LIN {X 0,Y 742.952,Z 751.201,A -85,B 0,C 180,E1 34860.975,E2 34860.975} C_VEL
LIN {X 0,Y 742.857,Z 676.201,A -85,B 0,C 180,E1 34860.963,E2 34860.963} C_VEL
LIN {X 0,Y 740.648,Z 678.554,A -85,B 0,C 180,E1 34860.677,E2 34860.677} C_VEL
LIN {X 0,Y 736.693,Z 689.627,A -85,B 0,C 180,E1 34860.154,E2 34860.154} C_VEL
LIN {X 0,Y 733.637,Z 695.78,A -85,B 0,C 180,E1 34859.741,E2 34859.741} C_VEL
LIN {X 0,Y 731.906,Z 697.683,A -85,B 0,C 180,E1 34859.503,E2 34859.503} C_VEL
LIN {X 0,Y 730.902,Z 697.691,A -85,B 0,C 180,E1 34859.356,E2 34859.356} C_VEL
LIN {X 0,Y 730.384,Z 754.623,A -85,B 0,C 180,E1 34856.592,E2 34856.592} C_VEL
LIN {X 0,Y 730.458,Z 758.053,A -85,B 0,C 180,E1 34856.45,E2 34856.45} C_VEL
LIN {X 0,Y 731.039,Z 764.29,A -85,B 0,C 180,E1 34856.361,E2 34856.361} C_VEL
LIN {X 0,Y 730.433,Z 1030.735,A -85,B 0,C 180,E1 34853.553,E2 34853.553} C_VEL
LIN {X 0,Y 730.302,Z 1066.289,A -85,B 0,C 180,E1 34853.15,E2 34853.15} C_VEL
LIN {X 0,Y 730.172,Z 1088.567,A -85,B 0,C 180,E1 34852.744,E2 34852.744} C_VEL
LIN {X 0,Y 729.954,Z 1109.789,A -85,B 0,C 180,E1 34852.212,E2 34852.212} C_VEL
LIN {X 0,Y 729.742,Z 1130.728,A -85,B 0,C 180,E1 34851.542,E2 34851.542} C_VEL
LIN {X 0,Y 729.516,Z 1150.772,A -85,B 0,C 180,E1 34850.749,E2 34850.749} C_VEL
LIN {X 0,Y 729.234,Z 1170.779,A -85,B 0,C 180,E1 34849.795,E2 34849.795} C_VEL
LIN {X 0,Y 728.966,Z 1190.488,A -85,B 0,C 180,E1 34848.678,E2 34848.678} C_VEL
LIN {X 0,Y 728.744,Z 1208.382,A -85,B 0,C 180,E1 34847.485,E2 34847.485} C_VEL
LIN {X 0,Y 728.539,Z 1225.234,A -85,B 0,C 180,E1 34846.176,E2 34846.176} C_VEL
LIN {X 0,Y 728.348,Z 1240.435,A -85,B 0,C 180,E1 34844.793,E2 34844.793} C_VEL
LIN {X 0,Y 728.19,Z 1254.18,A -85,B 0,C 180,E1 34843.336,E2 34843.336} C_VEL
LIN {X 0,Y 728.089,Z 1266.501,A -85,B 0,C 180,E1 34841.806,E2 34841.806} C_VEL
LIN {X 0,Y 728.01,Z 1276.879,A -85,B 0,C 180,E1 34840.284,E2 34840.284} C_VEL
LIN {X 0,Y 727.957,Z 1285.903,A -85,B 0,C 180,E1 34838.689,E2 34838.689} C_VEL
LIN {X 0,Y 727.931,Z 1293.551,A -85,B 0,C 180,E1 34837.021,E2 34837.021} C_VEL
LIN {X 0,Y 727.921,Z 1299.154,A -85,B 0,C 180,E1 34835.437,E2 34835.437} C_VEL
LIN {X 0,Y 727.911,Z 1303.638,A -85,B 0,C 180,E1 34833.701,E2 34833.701} C_VEL
LIN {X 0,Y 727.911,Z 1306.402,A -85,B 0,C 180,E1 34831.967,E2 34831.967} C_VEL
LIN {X 0,Y 727.9,Z 1307.418,A -85,B 0,C 180,E1 34830.314,E2 34830.314} C_VEL
LIN {X 0,Y 727.905,Z 1306.824,A -85,B 0,C 180,E1 34828.503,E2 34828.503} C_VEL
LIN {X 0,Y 727.917,Z 1304.577,A -85,B 0,C 180,E1 34826.77,E2 34826.77} C_VEL
LIN {X 0,Y 727.912,Z 1300.582,A -85,B 0,C 180,E1 34825.034,E2 34825.034} C_VEL
LIN {X 0,Y 727.917,Z 1295.067,A -85,B 0,C 180,E1 34823.373,E2 34823.373} C_VEL
LIN {X 0,Y 727.962,Z 1287.918,A -85,B 0,C 180,E1 34821.707,E2 34821.707} C_VEL
LIN {X 0,Y 728.002,Z 1278.375,A -85,B 0,C 180,E1 34819.954,E2 34819.954} C_VEL
LIN {X 0,Y 728.078,Z 1268.214,A -85,B 0,C 180,E1 34818.433,E2 34818.433} C_VEL
LIN {X 0,Y 728.182,Z 1256.277,A -85,B 0,C 180,E1 34816.904,E2 34816.904} C_VEL
LIN {X 0,Y 728.323,Z 1242.775,A -85,B 0,C 180,E1 34815.438,E2 34815.438} C_VEL
LIN {X 0,Y 728.489,Z 1228,A -85,B 0,C 180,E1 34814.066,E2 34814.066} C_VEL
LIN {X 0,Y 728.691,Z 1211.195,A -85,B 0,C 180,E1 34812.721,E2 34812.721} C_VEL
LIN {X 0,Y 728.938,Z 1193.096,A -85,B 0,C 180,E1 34811.484,E2 34811.484} C_VEL
LIN {X 0,Y 729.203,Z 1174.406,A -85,B 0,C 180,E1 34810.395,E2 34810.395} C_VEL
LIN {X 0,Y 729.459,Z 1154.716,A -85,B 0,C 180,E1 34809.425,E2 34809.425} C_VEL
LIN {X 0,Y 729.684,Z 1134.027,A -85,B 0,C 180,E1 34808.58,E2 34808.58} C_VEL
LIN {X 0,Y 729.94,Z 1112.649,A -85,B 0,C 180,E1 34807.87,E2 34807.87} C_VEL
LIN {X 0,Y 730.158,Z 1090.957,A -85,B 0,C 180,E1 34807.307,E2 34807.307} C_VEL
LIN {X 0,Y 730.291,Z 1068.704,A -85,B 0,C 180,E1 34806.888,E2 34806.888} C_VEL
LIN {X 0,Y 730.419,Z 1039.11,A -85,B 0,C 180,E1 34806.534,E2 34806.534} C_VEL
LIN {X 0,Y 731.027,Z 769.999,A -85,B 0,C 180,E1 34803.7,E2 34803.7} C_VEL
LIN {X 0,Y 730.771,Z 760.108,A -85,B 0,C 180,E1 34803.584,E2 34803.584} C_VEL
LIN {X 0,Y 730.359,Z 756.916,A -85,B 0,C 180,E1 34803.518,E2 34803.518} C_VEL
LIN {X 0,Y 730.883,Z 700.137,A -85,B 0,C 180,E1 34800.764,E2 34800.764} C_VEL
LIN {X 0,Y 730.937,Z 697.576,A -85,B 0,C 180,E1 34800.632,E2 34800.632} C_VEL
LIN {X 0,Y 732.166,Z 697.523,A -85,B 0,C 180,E1 34800.461,E2 34800.461} C_VEL
LIN {X 0,Y 734.394,Z 694.506,A -85,B 0,C 180,E1 34800.156,E2 34800.156} C_VEL
LIN {X 0,Y 737.903,Z 686.574,A -85,B 0,C 180,E1 34799.684,E2 34799.684} C_VEL
LIN {X 0,Y 740.949,Z 678.027,A -85,B 0,C 180,E1 34799.284,E2 34799.284} C_VEL
LIN {X 0,Y 742.946,Z 676.091,A -85,B 0,C 180,E1 34799.026,E2 34799.026} C_VEL
LIN {X 0,Y 743.089,Z 758.386,A -85,B 0,C 180,E1 34799.007,E2 34799.007} C_VEL
LIN {X 0,Y 744.031,Z 769.406,A -85,B 0,C 180,E1 34798.887,E2 34798.887} C_VEL
LIN {X 0,Y 745.78,Z 778.518,A -85,B 0,C 180,E1 34798.665,E2 34798.665} C_VEL
LIN {X 0,Y 748.328,Z 786.211,A -85,B 0,C 180,E1 34798.346,E2 34798.346} C_VEL
LIN {X 0,Y 750.526,Z 791.372,A -85,B 0,C 180,E1 34798.012,E2 34798.012} C_VEL
LIN {X 0,Y 751.455,Z 795.063,A -85,B 0,C 180,E1 34797.617,E2 34797.617} C_VEL
LIN {X 0,Y 751.184,Z 797.41,A -85,B 0,C 180,E1 34797.196,E2 34797.196} C_VEL
LIN {X 0,Y 749.781,Z 798.49,A -85,B 0,C 180,E1 34796.737,E2 34796.737} C_VEL
LIN {X 0,Y 747.366,Z 798.053,A -85,B 0,C 180,E1 34796.273,E2 34796.273} C_VEL
LIN {X 0,Y 744.248,Z 795.961,A -85,B 0,C 180,E1 34795.834,E2 34795.834} C_VEL
LIN {X 0,Y 740.757,Z 792.046,A -85,B 0,C 180,E1 34795.426,E2 34795.426} C_VEL
LIN {X 0,Y 736.905,Z 785.025,A -85,B 0,C 180,E1 34794.905,E2 34794.905} C_VEL
LIN {X 0,Y 733.978,Z 775.313,A -85,B 0,C 180,E1 34794.285,E2 34794.285} C_VEL
LIN {X 0,Y 732.165,Z 761.566,A -85,B 0,C 180,E1 34793.505,E2 34793.505} C_VEL
LIN {X 0,Y 731.75,Z 739.57,A -85,B 0,C 180,E1 34792.352,E2 34792.352} C_VEL
LIN {X 0,Y 732.362,Z 691.972,A -85,B 0,C 180,E1 34789.869,E2 34789.869} C_VEL
LIN {X 0,Y 732.889,Z 653.135,A -85,B 0,C 180,E1 34787.773,E2 34787.773} C_VEL
LIN {X 0,Y 728.341,Z 643.029,A -85,B 0,C 180,E1 34786.916,E2 34786.916} C_VEL
LIN {X 0,Y 728.135,Z 641.972,A -85,B 0,C 180,E1 34786.818,E2 34786.818} C_VEL
LIN {X 0,Y 728.143,Z 641.968,A -85,B 0,C 180,E1 34783.981,E2 34783.981} C_VEL
LIN {X 0,Y 728.163,Z 641.969,A -85,B 0,C 180,E1 34780.953,E2 34780.953} C_VEL
LIN {X 0,Y 728.159,Z 641.969,A -85,B 0,C 180,E1 34777.965,E2 34777.965} C_VEL
LIN {X 0,Y 728.159,Z 641.966,A -85,B 0,C 180,E1 34774.933,E2 34774.933} C_VEL
LIN {X 0,Y 728.147,Z 641.969,A -85,B 0,C 180,E1 34771.917,E2 34771.917} C_VEL
LIN {X 0,Y 728.156,Z 642.035,A -85,B 0,C 180,E1 34771.033,E2 34771.033} C_VEL
LIN {X 0,Y 730.274,Z 649.961,A -85,B 0,C 180,E1 34770.302,E2 34770.302} C_VEL
LIN {X 0,Y 729.837,Z 688.921,A -85,B 0,C 180,E1 34767.271,E2 34767.271} C_VEL
LIN {X 0,Y 729.783,Z 700.534,A -85,B 0,C 180,E1 34766.405,E2 34766.405} C_VEL
LIN {X 0,Y 731.037,Z 707.098,A -85,B 0,C 180,E1 34766.286,E2 34766.286} C_VEL
LIN {X 0,Y 730.396,Z 989.764,A -85,B 0,C 180,E1 34763.31,E2 34763.31} C_VEL
LIN {X 0,Y 730.277,Z 1013.096,A -85,B 0,C 180,E1 34762.995,E2 34762.995} C_VEL
LIN {X 0,Y 730.087,Z 1036.014,A -85,B 0,C 180,E1 34762.528,E2 34762.528} C_VEL
LIN {X 0,Y 729.907,Z 1056.833,A -85,B 0,C 180,E1 34761.961,E2 34761.961} C_VEL
LIN {X 0,Y 729.659,Z 1077.192,A -85,B 0,C 180,E1 34761.256,E2 34761.256} C_VEL
LIN {X 0,Y 729.394,Z 1097.987,A -85,B 0,C 180,E1 34760.377,E2 34760.377} C_VEL
LIN {X 0,Y 729.169,Z 1116.946,A -85,B 0,C 180,E1 34759.423,E2 34759.423} C_VEL
LIN {X 0,Y 728.918,Z 1135.28,A -85,B 0,C 180,E1 34758.332,E2 34758.332} C_VEL
LIN {X 0,Y 728.671,Z 1152.67,A -85,B 0,C 180,E1 34757.123,E2 34757.123} C_VEL
LIN {X 0,Y 728.462,Z 1169.367,A -85,B 0,C 180,E1 34755.77,E2 34755.77} C_VEL
LIN {X 0,Y 728.309,Z 1184.031,A -85,B 0,C 180,E1 34754.388,E2 34754.388} C_VEL
LIN {X 0,Y 728.18,Z 1197.276,A -85,B 0,C 180,E1 34752.934,E2 34752.934} C_VEL
LIN {X 0,Y 728.069,Z 1209.071,A -85,B 0,C 180,E1 34751.406,E2 34751.406} C_VEL
LIN {X 0,Y 728,Z 1219.955,A -85,B 0,C 180,E1 34749.726,E2 34749.726} C_VEL
LIN {X 0,Y 727.953,Z 1228.483,A -85,B 0,C 180,E1 34748.133,E2 34748.133} C_VEL
LIN {X 0,Y 727.921,Z 1235.5,A -85,B 0,C 180,E1 34746.467,E2 34746.467} C_VEL
LIN {X 0,Y 727.914,Z 1241.076,A -85,B 0,C 180,E1 34744.728,E2 34744.728} C_VEL
LIN {X 0,Y 727.898,Z 1244.794,A -85,B 0,C 180,E1 34743.071,E2 34743.071} C_VEL
LIN {X 0,Y 727.907,Z 1246.91,A -85,B 0,C 180,E1 34741.338,E2 34741.338} C_VEL
LIN {X 0,Y 727.917,Z 1247.386,A -85,B 0,C 180,E1 34739.528,E2 34739.528} C_VEL
LIN {X 0,Y 727.903,Z 1246.183,A -85,B 0,C 180,E1 34737.796,E2 34737.796} C_VEL
LIN {X 0,Y 727.901,Z 1243.24,A -85,B 0,C 180,E1 34736.062,E2 34736.062} C_VEL
LIN {X 0,Y 727.919,Z 1238.796,A -85,B 0,C 180,E1 34734.403,E2 34734.403} C_VEL
LIN {X 0,Y 727.94,Z 1232.782,A -85,B 0,C 180,E1 34732.74,E2 34732.74} C_VEL
LIN {X 0,Y 727.968,Z 1225.299,A -85,B 0,C 180,E1 34731.151,E2 34731.151} C_VEL
LIN {X 0,Y 728.024,Z 1215.515,A -85,B 0,C 180,E1 34729.459,E2 34729.459} C_VEL
LIN {X 0,Y 728.118,Z 1204.447,A -85,B 0,C 180,E1 34727.871,E2 34727.871} C_VEL
LIN {X 0,Y 728.169,Z 1198.333,A -85,B 0,C 180,E1 34727.101,E2 34727.101} C_VEL
LIN {X 0,Y 727.25,Z 1194.197,A -85,B 0,C 180,E1 34726.589,E2 34726.589} C_VEL
LIN {X 0,Y 721.178,Z 1182.848,A -85,B 0,C 180,E1 34725.25,E2 34725.25} C_VEL
LIN {X 0,Y 720.487,Z 1178.753,A -85,B 0,C 180,E1 34724.834,E2 34724.834} C_VEL
LIN {X 0,Y 720.715,Z 1163.654,A -85,B 0,C 180,E1 34723.469,E2 34723.469} C_VEL
LIN {X 0,Y 721.001,Z 1147.118,A -85,B 0,C 180,E1 34722.18,E2 34722.18} C_VEL
LIN {X 0,Y 721.273,Z 1129.813,A -85,B 0,C 180,E1 34721.029,E2 34721.029} C_VEL
LIN {X 0,Y 721.585,Z 1110.77,A -85,B 0,C 180,E1 34719.943,E2 34719.943} C_VEL
LIN {X 0,Y 721.934,Z 1090.961,A -85,B 0,C 180,E1 34718.988,E2 34718.988} C_VEL
LIN {X 0,Y 722.229,Z 1070.731,A -85,B 0,C 180,E1 34718.178,E2 34718.178} C_VEL
LIN {X 0,Y 722.504,Z 1049.773,A -85,B 0,C 180,E1 34717.502,E2 34717.502} C_VEL
LIN {X 0,Y 722.771,Z 1027.33,A -85,B 0,C 180,E1 34716.94,E2 34716.94} C_VEL
LIN {X 0,Y 722.959,Z 1005.469,A -85,B 0,C 180,E1 34716.543,E2 34716.543} C_VEL
LIN {X 0,Y 723.116,Z 963.006,A -85,B 0,C 180,E1 34716.067,E2 34716.067} C_VEL
LIN {X 0,Y 723.828,Z 707.229,A -85,B 0,C 180,E1 34713.343,E2 34713.343} C_VEL
LIN {X 0,Y 722.222,Z 700.036,A -85,B 0,C 180,E1 34713.192,E2 34713.192} C_VEL
LIN {X 0,Y 722.727,Z 662.539,A -85,B 0,C 180,E1 34710.265,E2 34710.265} C_VEL
LIN {X 0,Y 722.701,Z 651.507,A -85,B 0,C 180,E1 34709.381,E2 34709.381} C_VEL
LIN {X 0,Y 720.204,Z 642.955,A -85,B 0,C 180,E1 34708.555,E2 34708.555} C_VEL
LIN {X 0,Y 720.218,Z 642.961,A -85,B 0,C 180,E1 34705.691,E2 34705.691} C_VEL
LIN {X 0,Y 720.202,Z 642.954,A -85,B 0,C 180,E1 34702.748,E2 34702.748} C_VEL
LIN {X 0,Y 720.209,Z 642.953,A -85,B 0,C 180,E1 34699.791,E2 34699.791} C_VEL
LIN {X 0,Y 720.218,Z 642.959,A -85,B 0,C 180,E1 34696.792,E2 34696.792} C_VEL
LIN {X 0,Y 720.215,Z 642.952,A -85,B 0,C 180,E1 34693.786,E2 34693.786} C_VEL
LIN {X 0,Y 720.212,Z 642.951,A -85,B 0,C 180,E1 34690.709,E2 34690.709} C_VEL
LIN {X 0,Y 720.221,Z 642.954,A -85,B 0,C 180,E1 34687.652,E2 34687.652} C_VEL
LIN {X 0,Y 720.199,Z 642.956,A -85,B 0,C 180,E1 34684.697,E2 34684.697} C_VEL
LIN {X 0,Y 720.196,Z 642.952,A -85,B 0,C 180,E1 34681.823,E2 34681.823} C_VEL
LIN {X 0,Y 720.212,Z 642.959,A -85,B 0,C 180,E1 34678.891,E2 34678.891} C_VEL
LIN {X 0,Y 720.215,Z 642.952,A -85,B 0,C 180,E1 34675.934,E2 34675.934} C_VEL
LIN {X 0,Y 720.222,Z 642.949,A -85,B 0,C 180,E1 34672.876,E2 34672.876} C_VEL
LIN {X 0,Y 720.221,Z 642.953,A -85,B 0,C 180,E1 34669.732,E2 34669.732} C_VEL
LIN {X 0,Y 720.211,Z 642.955,A -85,B 0,C 180,E1 34666.785,E2 34666.785} C_VEL
LIN {X 0,Y 720.202,Z 642.95,A -85,B 0,C 180,E1 34663.816,E2 34663.816} C_VEL
LIN {X 0,Y 720.213,Z 642.955,A -85,B 0,C 180,E1 34660.884,E2 34660.884} C_VEL
LIN {X 0,Y 720.212,Z 642.953,A -85,B 0,C 180,E1 34657.901,E2 34657.901} C_VEL
LIN {X 0,Y 720.208,Z 642.95,A -85,B 0,C 180,E1 34655.019,E2 34655.019} C_VEL
LIN {X 0,Y 720.214,Z 642.955,A -85,B 0,C 180,E1 34651.99,E2 34651.99} C_VEL
LIN {X 0,Y 720.217,Z 642.952,A -85,B 0,C 180,E1 34649.047,E2 34649.047} C_VEL
LIN {X 0,Y 720.208,Z 642.949,A -85,B 0,C 180,E1 34646.021,E2 34646.021} C_VEL
LIN {X 0,Y 720.201,Z 642.955,A -85,B 0,C 180,E1 34643.061,E2 34643.061} C_VEL
LIN {X 0,Y 720.198,Z 642.954,A -85,B 0,C 180,E1 34640.25,E2 34640.25} C_VEL
LIN {X 0,Y 720.208,Z 642.952,A -85,B 0,C 180,E1 34637.33,E2 34637.33} C_VEL
LIN {X 0,Y 720.219,Z 642.959,A -85,B 0,C 180,E1 34634.377,E2 34634.377} C_VEL
LIN {X 0,Y 720.214,Z 642.952,A -85,B 0,C 180,E1 34631.38,E2 34631.38} C_VEL
LIN {X 0,Y 720.209,Z 642.951,A -85,B 0,C 180,E1 34628.329,E2 34628.329} C_VEL
LIN {X 0,Y 720.221,Z 642.956,A -85,B 0,C 180,E1 34625.388,E2 34625.388} C_VEL
LIN {X 0,Y 720.199,Z 642.954,A -85,B 0,C 180,E1 34622.465,E2 34622.465} C_VEL
LIN {X 0,Y 720.203,Z 642.953,A -85,B 0,C 180,E1 34619.554,E2 34619.554} C_VEL
LIN {X 0,Y 720.213,Z 642.96,A -85,B 0,C 180,E1 34616.552,E2 34616.552} C_VEL
LIN {X 0,Y 720.215,Z 642.951,A -85,B 0,C 180,E1 34613.546,E2 34613.546} C_VEL
LIN {X 0,Y 720.221,Z 642.95,A -85,B 0,C 180,E1 34610.519,E2 34610.519} C_VEL
LIN {X 0,Y 720.214,Z 642.957,A -85,B 0,C 180,E1 34607.462,E2 34607.462} C_VEL
LIN {X 0,Y 720.199,Z 642.956,A -85,B 0,C 180,E1 34604.586,E2 34604.586} C_VEL
LIN {X 0,Y 720.197,Z 642.956,A -85,B 0,C 180,E1 34601.684,E2 34601.684} C_VEL
LIN {X 0,Y 720.209,Z 643.023,A -85,B 0,C 180,E1 34599.75,E2 34599.75} C_VEL
LIN {X 0,Y 723.542,Z 653.303,A -85,B 0,C 180,E1 34598.859,E2 34598.859} C_VEL
LIN {X 0,Y 723.026,Z 697.05,A -85,B 0,C 180,E1 34595.869,E2 34595.869} C_VEL
LIN {X 0,Y 722.245,Z 740.336,A -85,B 0,C 180,E1 34592.962,E2 34592.962} C_VEL
LIN {X 0,Y 721.605,Z 784.471,A -85,B 0,C 180,E1 34590.061,E2 34590.061} C_VEL
LIN {X 0,Y 720.989,Z 830.529,A -85,B 0,C 180,E1 34587.057,E2 34587.057} C_VEL
LIN {X 0,Y 720.633,Z 881.161,A -85,B 0,C 180,E1 34583.888,E2 34583.888} C_VEL
LIN {X 0,Y 720.605,Z 891.749,A -85,B 0,C 180,E1 34583.256,E2 34583.256} C_VEL
LIN {X 0,Y 720.898,Z 904.834,A -85,B 0,C 180,E1 34583.119,E2 34583.119} C_VEL
LIN {X 0,Y 720.691,Z 1032.433,A -85,B 0,C 180,E1 34581.826,E2 34581.826} C_VEL
LIN {X 0,Y 720.626,Z 1046.219,A -85,B 0,C 180,E1 34581.581,E2 34581.581} C_VEL
LIN {X 0,Y 720.548,Z 1061.079,A -85,B 0,C 180,E1 34581.192,E2 34581.192} C_VEL
LIN {X 0,Y 720.428,Z 1077.241,A -85,B 0,C 180,E1 34580.6,E2 34580.6} C_VEL
LIN {X 0,Y 720.304,Z 1090.348,A -85,B 0,C 180,E1 34579.967,E2 34579.967} C_VEL
LIN {X 0,Y 720.224,Z 1102.147,A -85,B 0,C 180,E1 34579.263,E2 34579.263} C_VEL
LIN {X 0,Y 720.136,Z 1112.636,A -85,B 0,C 180,E1 34578.506,E2 34578.506} C_VEL
LIN {X 0,Y 720.064,Z 1121.875,A -85,B 0,C 180,E1 34577.704,E2 34577.704} C_VEL
LIN {X 0,Y 720.002,Z 1130.631,A -85,B 0,C 180,E1 34576.79,E2 34576.79} C_VEL
LIN {X 0,Y 719.965,Z 1138.65,A -85,B 0,C 180,E1 34575.76,E2 34575.76} C_VEL
LIN {X 0,Y 719.935,Z 1146.365,A -85,B 0,C 180,E1 34574.477,E2 34574.477} C_VEL
LIN {X 0,Y 719.922,Z 1151.651,A -85,B 0,C 180,E1 34573.248,E2 34573.248} C_VEL
LIN {X 0,Y 719.917,Z 1154.986,A -85,B 0,C 180,E1 34572.106,E2 34572.106} C_VEL
LIN {X 0,Y 719.918,Z 1156.891,A -85,B 0,C 180,E1 34570.969,E2 34570.969} C_VEL
LIN {X 0,Y 719.916,Z 1157.432,A -85,B 0,C 180,E1 34569.756,E2 34569.756} C_VEL
LIN {X 0,Y 719.916,Z 1156.202,A -85,B 0,C 180,E1 34568.386,E2 34568.386} C_VEL
LIN {X 0,Y 719.92,Z 1153.128,A -85,B 0,C 180,E1 34567.101,E2 34567.101} C_VEL
LIN {X 0,Y 719.925,Z 1148.55,A -85,B 0,C 180,E1 34565.899,E2 34565.899} C_VEL
LIN {X 0,Y 719.944,Z 1143.158,A -85,B 0,C 180,E1 34564.86,E2 34564.86} C_VEL
LIN {X 0,Y 719.976,Z 1136.274,A -85,B 0,C 180,E1 34563.822,E2 34563.822} C_VEL
LIN {X 0,Y 720.031,Z 1127.684,A -85,B 0,C 180,E1 34562.786,E2 34562.786} C_VEL
LIN {X 0,Y 720.119,Z 1115.936,A -85,B 0,C 180,E1 34561.671,E2 34561.671} C_VEL
LIN {X 0,Y 720.202,Z 1104.974,A -85,B 0,C 180,E1 34560.835,E2 34560.835} C_VEL
LIN {X 0,Y 720.291,Z 1093.518,A -85,B 0,C 180,E1 34560.119,E2 34560.119} C_VEL
LIN {X 0,Y 720.363,Z 1081.901,A -85,B 0,C 180,E1 34559.523,E2 34559.523} C_VEL
LIN {X 0,Y 720.485,Z 1069.428,A -85,B 0,C 180,E1 34559.006,E2 34559.006} C_VEL
LIN {X 0,Y 720.573,Z 1056.573,A -85,B 0,C 180,E1 34558.589,E2 34558.589} C_VEL
LIN {X 0,Y 720.644,Z 1042.354,A -85,B 0,C 180,E1 34558.248,E2 34558.248} C_VEL
LIN {X 0,Y 720.719,Z 1025.411,A -85,B 0,C 180,E1 34557.994,E2 34557.994} C_VEL
LIN {X 0,Y 720.682,Z 892.464,A -85,B 0,C 180,E1 34556.663,E2 34556.663} C_VEL
LIN {X 0,Y 720.553,Z 890.779,A -85,B 0,C 180,E1 34556.619,E2 34556.619} C_VEL
LIN {X 0,Y 720.891,Z 843.506,A -85,B 0,C 180,E1 34553.669,E2 34553.669} C_VEL
LIN {X 0,Y 721.186,Z 820.191,A -85,B 0,C 180,E1 34552.151,E2 34552.151} C_VEL
LIN {X 0,Y 722.359,Z 776.041,A -85,B 0,C 180,E1 34549.149,E2 34549.149} C_VEL
LIN {X 0,Y 723.806,Z 731.519,A -85,B 0,C 180,E1 34546.051,E2 34546.051} C_VEL
LIN {X 0,Y 725.105,Z 696.365,A -85,B 0,C 180,E1 34543.538,E2 34543.538} C_VEL
LIN {X 0,Y 725.937,Z 658.569,A -85,B 0,C 180,E1 34540.696,E2 34540.696} C_VEL
LIN {X 0,Y 725.651,Z 656.599,A -85,B 0,C 180,E1 34540.521,E2 34540.521} C_VEL
LIN {X 0,Y 721.022,Z 645.626,A -85,B 0,C 180,E1 34539.291,E2 34539.291} C_VEL
LIN {X 0,Y 720.203,Z 642.961,A -85,B 0,C 180,E1 34538.971,E2 34538.971} C_VEL
LIN {X 0,Y 720.199,Z 642.957,A -85,B 0,C 180,E1 34536.084,E2 34536.084} C_VEL
LIN {X 0,Y 720.202,Z 642.952,A -85,B 0,C 180,E1 34533.178,E2 34533.178} C_VEL
LIN {X 0,Y 720.21,Z 642.959,A -85,B 0,C 180,E1 34530.197,E2 34530.197} C_VEL
LIN {X 0,Y 720.22,Z 642.948,A -85,B 0,C 180,E1 34527.218,E2 34527.218} C_VEL
LIN {X 0,Y 720.217,Z 642.96,A -85,B 0,C 180,E1 34524.135,E2 34524.135} C_VEL
LIN {X 0,Y 720.222,Z 642.948,A -85,B 0,C 180,E1 34521.025,E2 34521.025} C_VEL
LIN {X 0,Y 720.22,Z 642.958,A -85,B 0,C 180,E1 34517.89,E2 34517.89} C_VEL
LIN {X 0,Y 720.216,Z 642.951,A -85,B 0,C 180,E1 34514.811,E2 34514.811} C_VEL
LIN {X 0,Y 720.233,Z 643.173,A -85,B 0,C 180,E1 34512.95,E2 34512.95} C_VEL
LIN {X 0,Y 724.99,Z 654.917,A -85,B 0,C 180,E1 34512.006,E2 34512.006} C_VEL
LIN {X 0,Y 723.849,Z 704.769,A -85,B 0,C 180,E1 34509.449,E2 34509.449} C_VEL
LIN {X 0,Y 723.616,Z 756.565,A -85,B 0,C 180,E1 34506.896,E2 34506.896} C_VEL
LIN {X 0,Y 725.456,Z 773.802,A -85,B 0,C 180,E1 34505.996,E2 34505.996} C_VEL
LIN {X 0,Y 728.528,Z 785.626,A -85,B 0,C 180,E1 34505.319,E2 34505.319} C_VEL
LIN {X 0,Y 732.679,Z 794.35,A -85,B 0,C 180,E1 34504.759,E2 34504.759} C_VEL
LIN {X 0,Y 737.283,Z 800.328,A -85,B 0,C 180,E1 34504.318,E2 34504.318} C_VEL
LIN {X 0,Y 741.214,Z 803.709,A -85,B 0,C 180,E1 34503.939,E2 34503.939} C_VEL
LIN {X 0,Y 744.72,Z 805.498,A -85,B 0,C 180,E1 34503.511,E2 34503.511} C_VEL
LIN {X 0,Y 747.247,Z 805.772,A -85,B 0,C 180,E1 34503.087,E2 34503.087} C_VEL
LIN {X 0,Y 748.979,Z 804.654,A -85,B 0,C 180,E1 34502.606,E2 34502.606} C_VEL
LIN {X 0,Y 749.398,Z 802.128,A -85,B 0,C 180,E1 34502.141,E2 34502.141} C_VEL
LIN {X 0,Y 748.459,Z 798.545,A -85,B 0,C 180,E1 34501.735,E2 34501.735} C_VEL
LIN {X 0,Y 746.027,Z 793.391,A -85,B 0,C 180,E1 34501.366,E2 34501.366} C_VEL
LIN {X 0,Y 742.954,Z 785.217,A -85,B 0,C 180,E1 34500.975,E2 34500.975} C_VEL
LIN {X 0,Y 740.745,Z 775.804,A -85,B 0,C 180,E1 34500.689,E2 34500.689} C_VEL
LIN {X 0,Y 739.376,Z 765.011,A -85,B 0,C 180,E1 34500.51,E2 34500.51} C_VEL
LIN {X 0,Y 738.869,Z 752.866,A -85,B 0,C 180,E1 34500.444,E2 34500.444} C_VEL
LIN {X 0,Y 738.837,Z 696.94,A -85,B 0,C 180,E1 34500.439,E2 34500.439} C_VEL
LIN {X 0,Y 735.629,Z 702.763,A -85,B 0,C 180,E1 34500.011,E2 34500.011} C_VEL
LIN {X 0,Y 733.171,Z 705.566,A -85,B 0,C 180,E1 34499.677,E2 34499.677} C_VEL
LIN {X 0,Y 729.153,Z 717.357,A -85,B 0,C 180,E1 34499.118,E2 34499.118} C_VEL
LIN {X 0,Y 726.072,Z 723.927,A -85,B 0,C 180,E1 34498.679,E2 34498.679} C_VEL
LIN {X 0,Y 724.4,Z 725.949,A -85,B 0,C 180,E1 34498.436,E2 34498.436} C_VEL
LIN {X 0,Y 723.378,Z 726.043,A -85,B 0,C 180,E1 34498.277,E2 34498.277} C_VEL
LIN {X 0,Y 723.091,Z 757.88,A -85,B 0,C 180,E1 34496.743,E2 34496.743} C_VEL
LIN {X 0,Y 723.867,Z 764.998,A -85,B 0,C 180,E1 34496.635,E2 34496.635} C_VEL
LIN {X 0,Y 723.094,Z 1032.343,A -85,B 0,C 180,E1 34493.79,E2 34493.79} C_VEL
LIN {X 0,Y 722.934,Z 1066.626,A -85,B 0,C 180,E1 34493.394,E2 34493.394} C_VEL
LIN {X 0,Y 722.766,Z 1088.808,A -85,B 0,C 180,E1 34492.985,E2 34492.985} C_VEL
LIN {X 0,Y 722.492,Z 1110.581,A -85,B 0,C 180,E1 34492.431,E2 34492.431} C_VEL
LIN {X 0,Y 722.209,Z 1131.856,A -85,B 0,C 180,E1 34491.736,E2 34491.736} C_VEL
LIN {X 0,Y 721.93,Z 1151.747,A -85,B 0,C 180,E1 34490.935,E2 34490.935} C_VEL
LIN {X 0,Y 721.579,Z 1171.589,A -85,B 0,C 180,E1 34489.971,E2 34489.971} C_VEL
LIN {X 0,Y 721.248,Z 1191.156,A -85,B 0,C 180,E1 34488.844,E2 34488.844} C_VEL
LIN {X 0,Y 720.962,Z 1208.945,A -85,B 0,C 180,E1 34487.639,E2 34487.639} C_VEL
LIN {X 0,Y 720.689,Z 1226.17,A -85,B 0,C 180,E1 34486.274,E2 34486.274} C_VEL
LIN {X 0,Y 720.455,Z 1241.25,A -85,B 0,C 180,E1 34484.876,E2 34484.876} C_VEL
LIN {X 0,Y 720.264,Z 1254.889,A -85,B 0,C 180,E1 34483.404,E2 34483.404} C_VEL
LIN {X 0,Y 720.127,Z 1267.654,A -85,B 0,C 180,E1 34481.776,E2 34481.776} C_VEL
LIN {X 0,Y 720.032,Z 1277.883,A -85,B 0,C 180,E1 34480.237,E2 34480.237} C_VEL
LIN {X 0,Y 719.968,Z 1287.125,A -85,B 0,C 180,E1 34478.545,E2 34478.545} C_VEL
LIN {X 0,Y 719.924,Z 1294.47,A -85,B 0,C 180,E1 34476.859,E2 34476.859} C_VEL
LIN {X 0,Y 719.924,Z 1300.161,A -85,B 0,C 180,E1 34475.178,E2 34475.178} C_VEL
LIN {X 0,Y 719.916,Z 1304.43,A -85,B 0,C 180,E1 34473.343,E2 34473.343} C_VEL
LIN {X 0,Y 719.908,Z 1306.762,A -85,B 0,C 180,E1 34471.591,E2 34471.591} C_VEL
LIN {X 0,Y 719.902,Z 1307.44,A -85,B 0,C 180,E1 34469.76,E2 34469.76} C_VEL
LIN {X 0,Y 719.914,Z 1306.477,A -85,B 0,C 180,E1 34468.089,E2 34468.089} C_VEL
LIN {X 0,Y 719.913,Z 1303.794,A -85,B 0,C 180,E1 34466.336,E2 34466.336} C_VEL
LIN {X 0,Y 719.923,Z 1299.398,A -85,B 0,C 180,E1 34464.58,E2 34464.58} C_VEL
LIN {X 0,Y 719.935,Z 1293.851,A -85,B 0,C 180,E1 34462.979,E2 34462.979} C_VEL
LIN {X 0,Y 719.971,Z 1286.302,A -85,B 0,C 180,E1 34461.292,E2 34461.292} C_VEL
LIN {X 0,Y 720.043,Z 1276.859,A -85,B 0,C 180,E1 34459.599,E2 34459.599} C_VEL
LIN {X 0,Y 720.143,Z 1266.481,A -85,B 0,C 180,E1 34458.059,E2 34458.059} C_VEL
LIN {X 0,Y 720.288,Z 1253.46,A -85,B 0,C 180,E1 34456.431,E2 34456.431} C_VEL
LIN {X 0,Y 720.476,Z 1239.568,A -85,B 0,C 180,E1 34454.957,E2 34454.957} C_VEL
LIN {X 0,Y 720.716,Z 1223.698,A -85,B 0,C 180,E1 34453.517,E2 34453.517} C_VEL
LIN {X 0,Y 720.985,Z 1207.194,A -85,B 0,C 180,E1 34452.235,E2 34452.235} C_VEL
LIN {X 0,Y 721.279,Z 1189.797,A -85,B 0,C 180,E1 34451.071,E2 34451.071} C_VEL
LIN {X 0,Y 721.595,Z 1170.382,A -85,B 0,C 180,E1 34449.966,E2 34449.966} C_VEL
LIN {X 0,Y 721.942,Z 1150.725,A -85,B 0,C 180,E1 34449.02,E2 34449.02} C_VEL
LIN {X 0,Y 722.235,Z 1130.675,A -85,B 0,C 180,E1 34448.22,E2 34448.22} C_VEL
LIN {X 0,Y 722.498,Z 1109.724,A -85,B 0,C 180,E1 34447.544,E2 34447.544} C_VEL
LIN {X 0,Y 722.78,Z 1087.209,A -85,B 0,C 180,E1 34446.981,E2 34446.981} C_VEL
LIN {X 0,Y 722.961,Z 1064.711,A -85,B 0,C 180,E1 34446.577,E2 34446.577} C_VEL
LIN {X 0,Y 723.149,Z 1012.39,A -85,B 0,C 180,E1 34446,E2 34446} C_VEL
LIN {X 0,Y 723.815,Z 762.622,A -85,B 0,C 180,E1 34443.338,E2 34443.338} C_VEL
LIN {X 0,Y 723.015,Z 757.294,A -85,B 0,C 180,E1 34443.246,E2 34443.246} C_VEL
LIN {X 0,Y 723.463,Z 725.947,A -85,B 0,C 180,E1 34441.701,E2 34441.701} C_VEL
LIN {X 0,Y 724.65,Z 725.761,A -85,B 0,C 180,E1 34441.527,E2 34441.527} C_VEL
LIN {X 0,Y 726.867,Z 722.498,A -85,B 0,C 180,E1 34441.207,E2 34441.207} C_VEL
LIN {X 0,Y 730.325,Z 714.251,A -85,B 0,C 180,E1 34440.717,E2 34440.717} C_VEL
LIN {X 0,Y 733.401,Z 705.123,A -85,B 0,C 180,E1 34440.291,E2 34440.291} C_VEL
LIN {X 0,Y 736.017,Z 702.197,A -85,B 0,C 180,E1 34439.936,E2 34439.936} C_VEL
LIN {X 0,Y 738.861,Z 696.889,A -85,B 0,C 180,E1 34439.558,E2 34439.558} C_VEL
LIN {X 0,Y 739.005,Z 758.817,A -85,B 0,C 180,E1 34439.539,E2 34439.539} C_VEL
LIN {X 0,Y 739.947,Z 770.523,A -85,B 0,C 180,E1 34439.415,E2 34439.415} C_VEL
LIN {X 0,Y 741.684,Z 780.413,A -85,B 0,C 180,E1 34439.188,E2 34439.188} C_VEL
LIN {X 0,Y 744.225,Z 789.028,A -85,B 0,C 180,E1 34438.862,E2 34438.862} C_VEL
LIN {X 0,Y 747.505,Z 796.372,A -85,B 0,C 180,E1 34438.442,E2 34438.442} C_VEL
LIN {X 0,Y 749.095,Z 800.498,A -85,B 0,C 180,E1 34438.067,E2 34438.067} C_VEL
LIN {X 0,Y 749.363,Z 803.545,A -85,B 0,C 180,E1 34437.632,E2 34437.632} C_VEL
LIN {X 0,Y 748.372,Z 805.322,A -85,B 0,C 180,E1 34437.183,E2 34437.183} C_VEL
LIN {X 0,Y 746.261,Z 805.81,A -85,B 0,C 180,E1 34436.729,E2 34436.729} C_VEL
LIN {X 0,Y 743.028,Z 804.796,A -85,B 0,C 180,E1 34436.268,E2 34436.268} C_VEL
LIN {X 0,Y 739,Z 801.998,A -85,B 0,C 180,E1 34435.839,E2 34435.839} C_VEL
LIN {X 0,Y 734.152,Z 796.509,A -85,B 0,C 180,E1 34435.349,E2 34435.349} C_VEL
LIN {X 0,Y 730.13,Z 789.023,A -85,B 0,C 180,E1 34434.791,E2 34434.791} C_VEL
LIN {X 0,Y 727.065,Z 778.893,A -85,B 0,C 180,E1 34434.136,E2 34434.136} C_VEL
LIN {X 0,Y 725.187,Z 765.117,A -85,B 0,C 180,E1 34433.343,E2 34433.343} C_VEL
LIN {X 0,Y 724.726,Z 744.138,A -85,B 0,C 180,E1 34432.223,E2 34432.223} C_VEL
LIN {X 0,Y 725.487,Z 696.721,A -85,B 0,C 180,E1 34429.729,E2 34429.729} C_VEL
LIN {X 0,Y 726.162,Z 656.975,A -85,B 0,C 180,E1 34427.566,E2 34427.566} C_VEL
LIN {X 0,Y 720.262,Z 643.284,A -85,B 0,C 180,E1 34426.403,E2 34426.403} C_VEL
LIN {X 0,Y 720.22,Z 642.959,A -85,B 0,C 180,E1 34426.329,E2 34426.329} C_VEL
LIN {X 0,Y 720.224,Z 642.957,A -85,B 0,C 180,E1 34423.301,E2 34423.301} C_VEL
LIN {X 0,Y 720.204,Z 642.957,A -85,B 0,C 180,E1 34420.314,E2 34420.314} C_VEL
LIN {X 0,Y 720.197,Z 642.958,A -85,B 0,C 180,E1 34417.425,E2 34417.425} C_VEL
LIN {X 0,Y 720.214,Z 642.957,A -85,B 0,C 180,E1 34414.502,E2 34414.502} C_VEL
LIN {X 0,Y 720.217,Z 642.96,A -85,B 0,C 180,E1 34411.523,E2 34411.523} C_VEL
LIN {X 0,Y 720.232,Z 643.107,A -85,B 0,C 180,E1 34411.327,E2 34411.327} C_VEL
LIN {X 0,Y 722.864,Z 652.829,A -85,B 0,C 180,E1 34410.415,E2 34410.415} C_VEL
LIN {X 0,Y 722.326,Z 691.731,A -85,B 0,C 180,E1 34407.36,E2 34407.36} C_VEL
LIN {X 0,Y 722.292,Z 700.606,A -85,B 0,C 180,E1 34406.7,E2 34406.7} C_VEL
LIN {X 0,Y 723.859,Z 708.453,A -85,B 0,C 180,E1 34406.552,E2 34406.552} C_VEL
LIN {X 0,Y 723.047,Z 990.667,A -85,B 0,C 180,E1 34403.552,E2 34403.552} C_VEL
LIN {X 0,Y 722.896,Z 1013.581,A -85,B 0,C 180,E1 34403.235,E2 34403.235} C_VEL
LIN {X 0,Y 722.66,Z 1036.371,A -85,B 0,C 180,E1 34402.764,E2 34402.764} C_VEL
LIN {X 0,Y 722.432,Z 1057.199,A -85,B 0,C 180,E1 34402.19,E2 34402.19} C_VEL
LIN {X 0,Y 722.125,Z 1077.183,A -85,B 0,C 180,E1 34401.489,E2 34401.489} C_VEL
LIN {X 0,Y 721.798,Z 1098.001,A -85,B 0,C 180,E1 34400.601,E2 34400.601} C_VEL
LIN {X 0,Y 721.511,Z 1116.785,A -85,B 0,C 180,E1 34399.647,E2 34399.647} C_VEL
LIN {X 0,Y 721.192,Z 1135.004,A -85,B 0,C 180,E1 34398.554,E2 34398.554} C_VEL
LIN {X 0,Y 720.889,Z 1152.188,A -85,B 0,C 180,E1 34397.35,E2 34397.35} C_VEL
LIN {X 0,Y 720.638,Z 1168.448,A -85,B 0,C 180,E1 34396.029,E2 34396.029} C_VEL
LIN {X 0,Y 720.43,Z 1183.264,A -85,B 0,C 180,E1 34394.631,E2 34394.631} C_VEL
LIN {X 0,Y 720.256,Z 1196.583,A -85,B 0,C 180,E1 34393.16,E2 34393.16} C_VEL
LIN {X 0,Y 720.111,Z 1208.5,A -85,B 0,C 180,E1 34391.615,E2 34391.615} C_VEL
LIN {X 0,Y 720.035,Z 1219.038,A -85,B 0,C 180,E1 34389.996,E2 34389.996} C_VEL
LIN {X 0,Y 719.961,Z 1227.68,A -85,B 0,C 180,E1 34388.385,E2 34388.385} C_VEL
LIN {X 0,Y 719.932,Z 1234.897,A -85,B 0,C 180,E1 34386.7,E2 34386.7} C_VEL
LIN {X 0,Y 719.908,Z 1240.462,A -85,B 0,C 180,E1 34385.02,E2 34385.02} C_VEL
LIN {X 0,Y 719.906,Z 1244.322,A -85,B 0,C 180,E1 34383.344,E2 34383.344} C_VEL
LIN {X 0,Y 719.916,Z 1246.711,A -85,B 0,C 180,E1 34381.592,E2 34381.592} C_VEL
LIN {X 0,Y 719.915,Z 1247.474,A -85,B 0,C 180,E1 34379.841,E2 34379.841} C_VEL
LIN {X 0,Y 719.912,Z 1246.519,A -85,B 0,C 180,E1 34378.09,E2 34378.09} C_VEL
LIN {X 0,Y 719.914,Z 1243.871,A -85,B 0,C 180,E1 34376.337,E2 34376.337} C_VEL
LIN {X 0,Y 719.923,Z 1239.553,A -85,B 0,C 180,E1 34374.581,E2 34374.581} C_VEL
LIN {X 0,Y 719.945,Z 1233.724,A -85,B 0,C 180,E1 34372.9,E2 34372.9} C_VEL
LIN {X 0,Y 719.975,Z 1226.11,A -85,B 0,C 180,E1 34371.213,E2 34371.213} C_VEL
LIN {X 0,Y 720.04,Z 1217.158,A -85,B 0,C 180,E1 34369.6,E2 34369.6} C_VEL
LIN {X 0,Y 720.133,Z 1206.828,A -85,B 0,C 180,E1 34368.06,E2 34368.06} C_VEL
LIN {X 0,Y 720.272,Z 1194.55,A -85,B 0,C 180,E1 34366.513,E2 34366.513} C_VEL
LIN {X 0,Y 720.463,Z 1180.49,A -85,B 0,C 180,E1 34365.003,E2 34365.003} C_VEL
LIN {X 0,Y 720.487,Z 1178.753,A -85,B 0,C 180,E1 34364.834,E2 34364.834} C_VEL
LIN {X 0,Y 719.593,Z 1173.984,A -85,B 0,C 180,E1 34364.354,E2 34364.354} C_VEL
LIN {X 0,Y 713.717,Z 1161.147,A -85,B 0,C 180,E1 34363.082,E2 34363.082} C_VEL
LIN {X 0,Y 713.045,Z 1156.56,A -85,B 0,C 180,E1 34362.698,E2 34362.698} C_VEL
LIN {X 0,Y 713.383,Z 1139.486,A -85,B 0,C 180,E1 34361.448,E2 34361.448} C_VEL
LIN {X 0,Y 713.723,Z 1122.128,A -85,B 0,C 180,E1 34360.353,E2 34360.353} C_VEL
LIN {X 0,Y 714.128,Z 1103.416,A -85,B 0,C 180,E1 34359.339,E2 34359.339} C_VEL
LIN {X 0,Y 714.507,Z 1083.463,A -85,B 0,C 180,E1 34358.434,E2 34358.434} C_VEL
LIN {X 0,Y 714.85,Z 1063.351,A -85,B 0,C 180,E1 34357.681,E2 34357.681} C_VEL
LIN {X 0,Y 715.203,Z 1041.366,A -85,B 0,C 180,E1 34357.023,E2 34357.023} C_VEL
LIN {X 0,Y 715.469,Z 1019.525,A -85,B 0,C 180,E1 34356.525,E2 34356.525} C_VEL
LIN {X 0,Y 715.672,Z 997.208,A -85,B 0,C 180,E1 34356.179,E2 34356.179} C_VEL
LIN {X 0,Y 716.711,Z 708.918,A -85,B 0,C 180,E1 34353.076,E2 34353.076} C_VEL
LIN {X 0,Y 714.723,Z 700.034,A -85,B 0,C 180,E1 34352.888,E2 34352.888} C_VEL
LIN {X 0,Y 715.335,Z 663.104,A -85,B 0,C 180,E1 34349.973,E2 34349.973} C_VEL
LIN {X 0,Y 715.37,Z 654.441,A -85,B 0,C 180,E1 34349.272,E2 34349.272} C_VEL
LIN {X 0,Y 712.281,Z 643.943,A -85,B 0,C 180,E1 34348.258,E2 34348.258} C_VEL
LIN {X 0,Y 712.278,Z 643.943,A -85,B 0,C 180,E1 34345.156,E2 34345.156} C_VEL
LIN {X 0,Y 712.283,Z 643.947,A -85,B 0,C 180,E1 34342.058,E2 34342.058} C_VEL
LIN {X 0,Y 712.275,Z 643.943,A -85,B 0,C 180,E1 34339.037,E2 34339.037} C_VEL
LIN {X 0,Y 712.269,Z 643.941,A -85,B 0,C 180,E1 34335.982,E2 34335.982} C_VEL
LIN {X 0,Y 712.266,Z 643.946,A -85,B 0,C 180,E1 34332.997,E2 34332.997} C_VEL
LIN {X 0,Y 712.259,Z 643.944,A -85,B 0,C 180,E1 34330.118,E2 34330.118} C_VEL
LIN {X 0,Y 712.268,Z 643.94,A -85,B 0,C 180,E1 34327.233,E2 34327.233} C_VEL
LIN {X 0,Y 712.277,Z 643.947,A -85,B 0,C 180,E1 34324.225,E2 34324.225} C_VEL
LIN {X 0,Y 712.283,Z 643.94,A -85,B 0,C 180,E1 34321.199,E2 34321.199} C_VEL
LIN {X 0,Y 712.278,Z 643.938,A -85,B 0,C 180,E1 34318.053,E2 34318.053} C_VEL
LIN {X 0,Y 712.281,Z 643.941,A -85,B 0,C 180,E1 34314.926,E2 34314.926} C_VEL
LIN {X 0,Y 712.277,Z 643.949,A -85,B 0,C 180,E1 34311.888,E2 34311.888} C_VEL
LIN {X 0,Y 712.271,Z 643.94,A -85,B 0,C 180,E1 34308.885,E2 34308.885} C_VEL
LIN {X 0,Y 712.264,Z 643.941,A -85,B 0,C 180,E1 34305.888,E2 34305.888} C_VEL
LIN {X 0,Y 712.276,Z 643.946,A -85,B 0,C 180,E1 34302.981,E2 34302.981} C_VEL
LIN {X 0,Y 712.26,Z 643.942,A -85,B 0,C 180,E1 34300.026,E2 34300.026} C_VEL
LIN {X 0,Y 712.269,Z 643.942,A -85,B 0,C 180,E1 34297.097,E2 34297.097} C_VEL
LIN {X 0,Y 712.279,Z 643.946,A -85,B 0,C 180,E1 34294.107,E2 34294.107} C_VEL
LIN {X 0,Y 712.279,Z 643.94,A -85,B 0,C 180,E1 34291.047,E2 34291.047} C_VEL
LIN {X 0,Y 712.279,Z 643.939,A -85,B 0,C 180,E1 34287.909,E2 34287.909} C_VEL
LIN {X 0,Y 712.278,Z 643.942,A -85,B 0,C 180,E1 34284.766,E2 34284.766} C_VEL
LIN {X 0,Y 712.278,Z 643.944,A -85,B 0,C 180,E1 34281.761,E2 34281.761} C_VEL
LIN {X 0,Y 712.274,Z 643.938,A -85,B 0,C 180,E1 34278.667,E2 34278.667} C_VEL
LIN {X 0,Y 712.276,Z 643.939,A -85,B 0,C 180,E1 34275.61,E2 34275.61} C_VEL
LIN {X 0,Y 712.278,Z 643.948,A -85,B 0,C 180,E1 34272.603,E2 34272.603} C_VEL
LIN {X 0,Y 712.258,Z 643.942,A -85,B 0,C 180,E1 34269.679,E2 34269.679} C_VEL
LIN {X 0,Y 712.261,Z 643.943,A -85,B 0,C 180,E1 34266.768,E2 34266.768} C_VEL
LIN {X 0,Y 712.279,Z 643.947,A -85,B 0,C 180,E1 34263.847,E2 34263.847} C_VEL
LIN {X 0,Y 712.282,Z 643.939,A -85,B 0,C 180,E1 34260.828,E2 34260.828} C_VEL
LIN {X 0,Y 712.279,Z 643.936,A -85,B 0,C 180,E1 34257.764,E2 34257.764} C_VEL
LIN {X 0,Y 712.285,Z 643.942,A -85,B 0,C 180,E1 34254.647,E2 34254.647} C_VEL
LIN {X 0,Y 712.273,Z 643.945,A -85,B 0,C 180,E1 34251.651,E2 34251.651} C_VEL
LIN {X 0,Y 712.263,Z 643.941,A -85,B 0,C 180,E1 34248.681,E2 34248.681} C_VEL
LIN {X 0,Y 712.263,Z 643.948,A -85,B 0,C 180,E1 34245.721,E2 34245.721} C_VEL
LIN {X 0,Y 712.263,Z 643.945,A -85,B 0,C 180,E1 34242.881,E2 34242.881} C_VEL
LIN {X 0,Y 712.292,Z 643.996,A -85,B 0,C 180,E1 34240.091,E2 34240.091} C_VEL
LIN {X 0,Y 716.298,Z 656.224,A -85,B 0,C 180,E1 34239.018,E2 34239.018} C_VEL
LIN {X 0,Y 715.66,Z 700.214,A -85,B 0,C 180,E1 34235.985,E2 34235.985} C_VEL
LIN {X 0,Y 714.787,Z 744.914,A -85,B 0,C 180,E1 34232.967,E2 34232.967} C_VEL
LIN {X 0,Y 714.031,Z 789.031,A -85,B 0,C 180,E1 34230.042,E2 34230.042} C_VEL
LIN {X 0,Y 713.339,Z 833.687,A -85,B 0,C 180,E1 34227.101,E2 34227.101} C_VEL
LIN {X 0,Y 712.797,Z 877.907,A -85,B 0,C 180,E1 34224.25,E2 34224.25} C_VEL
LIN {X 0,Y 712.743,Z 891.726,A -85,B 0,C 180,E1 34223.405,E2 34223.405} C_VEL
LIN {X 0,Y 713.115,Z 901.377,A -85,B 0,C 180,E1 34223.3,E2 34223.3} C_VEL
LIN {X 0,Y 712.858,Z 1032.217,A -85,B 0,C 180,E1 34221.96,E2 34221.96} C_VEL
LIN {X 0,Y 712.788,Z 1045.187,A -85,B 0,C 180,E1 34221.731,E2 34221.731} C_VEL
LIN {X 0,Y 712.709,Z 1057.684,A -85,B 0,C 180,E1 34221.415,E2 34221.415} C_VEL
LIN {X 0,Y 712.601,Z 1069.447,A -85,B 0,C 180,E1 34221.025,E2 34221.025} C_VEL
LIN {X 0,Y 712.48,Z 1081.115,A -85,B 0,C 180,E1 34220.539,E2 34220.539} C_VEL
LIN {X 0,Y 712.374,Z 1092.006,A -85,B 0,C 180,E1 34219.985,E2 34219.985} C_VEL
LIN {X 0,Y 712.289,Z 1102.44,A -85,B 0,C 180,E1 34219.347,E2 34219.347} C_VEL
LIN {X 0,Y 712.19,Z 1112.362,A -85,B 0,C 180,E1 34218.623,E2 34218.623} C_VEL
LIN {X 0,Y 712.105,Z 1121.519,A -85,B 0,C 180,E1 34217.825,E2 34217.825} C_VEL
LIN {X 0,Y 712.035,Z 1129.603,A -85,B 0,C 180,E1 34216.983,E2 34216.983} C_VEL
LIN {X 0,Y 711.984,Z 1136.949,A -85,B 0,C 180,E1 34216.061,E2 34216.061} C_VEL
LIN {X 0,Y 711.953,Z 1143.424,A -85,B 0,C 180,E1 34215.059,E2 34215.059} C_VEL
LIN {X 0,Y 711.928,Z 1148.972,A -85,B 0,C 180,E1 34213.961,E2 34213.961} C_VEL
LIN {X 0,Y 711.918,Z 1153.705,A -85,B 0,C 180,E1 34212.656,E2 34212.656} C_VEL
LIN {X 0,Y 711.916,Z 1156.575,A -85,B 0,C 180,E1 34211.258,E2 34211.258} C_VEL
LIN {X 0,Y 711.916,Z 1157.419,A -85,B 0,C 180,E1 34210.094,E2 34210.094} C_VEL
LIN {X 0,Y 711.916,Z 1156.922,A -85,B 0,C 180,E1 34208.969,E2 34208.969} C_VEL
LIN {X 0,Y 711.918,Z 1155.084,A -85,B 0,C 180,E1 34207.83,E2 34207.83} C_VEL
LIN {X 0,Y 711.924,Z 1152.141,A -85,B 0,C 180,E1 34206.775,E2 34206.775} C_VEL
LIN {X 0,Y 711.932,Z 1147.943,A -85,B 0,C 180,E1 34205.723,E2 34205.723} C_VEL
LIN {X 0,Y 711.955,Z 1142.388,A -85,B 0,C 180,E1 34204.672,E2 34204.672} C_VEL
LIN {X 0,Y 712.002,Z 1134.748,A -85,B 0,C 180,E1 34203.543,E2 34203.543} C_VEL
LIN {X 0,Y 712.084,Z 1124.111,A -85,B 0,C 180,E1 34202.334,E2 34202.334} C_VEL
LIN {X 0,Y 712.171,Z 1114.362,A -85,B 0,C 180,E1 34201.448,E2 34201.448} C_VEL
LIN {X 0,Y 712.27,Z 1104.232,A -85,B 0,C 180,E1 34200.684,E2 34200.684} C_VEL
LIN {X 0,Y 712.371,Z 1093.341,A -85,B 0,C 180,E1 34200,E2 34200} C_VEL
LIN {X 0,Y 712.461,Z 1082.549,A -85,B 0,C 180,E1 34199.437,E2 34199.437} C_VEL
LIN {X 0,Y 712.595,Z 1071.304,A -85,B 0,C 180,E1 34198.955,E2 34198.955} C_VEL
LIN {X 0,Y 712.7,Z 1058.981,A -85,B 0,C 180,E1 34198.533,E2 34198.533} C_VEL
LIN {X 0,Y 712.779,Z 1045.889,A -85,B 0,C 180,E1 34198.194,E2 34198.194} C_VEL
LIN {X 0,Y 712.846,Z 1032.775,A -85,B 0,C 180,E1 34197.958,E2 34197.958} C_VEL
LIN {X 0,Y 712.961,Z 976.863,A -85,B 0,C 180,E1 34197.371,E2 34197.371} C_VEL
LIN {X 0,Y 712.894,Z 893.154,A -85,B 0,C 180,E1 34196.522,E2 34196.522} C_VEL
LIN {X 0,Y 712.695,Z 890.966,A -85,B 0,C 180,E1 34196.481,E2 34196.481} C_VEL
LIN {X 0,Y 713.024,Z 861.134,A -85,B 0,C 180,E1 34194.568,E2 34194.568} C_VEL
LIN {X 0,Y 714.031,Z 816.931,A -85,B 0,C 180,E1 34191.585,E2 34191.585} C_VEL
LIN {X 0,Y 715.348,Z 772.827,A -85,B 0,C 180,E1 34188.552,E2 34188.552} C_VEL
LIN {X 0,Y 716.914,Z 730.704,A -85,B 0,C 180,E1 34185.584,E2 34185.584} C_VEL
LIN {X 0,Y 718.254,Z 697.939,A -85,B 0,C 180,E1 34183.21,E2 34183.21} C_VEL
LIN {X 0,Y 719.268,Z 661.235,A -85,B 0,C 180,E1 34180.415,E2 34180.415} C_VEL
LIN {X 0,Y 713.407,Z 647.165,A -85,B 0,C 180,E1 34178.801,E2 34178.801} C_VEL
LIN {X 0,Y 712.271,Z 643.949,A -85,B 0,C 180,E1 34178.42,E2 34178.42} C_VEL
LIN {X 0,Y 712.277,Z 643.941,A -85,B 0,C 180,E1 34175.448,E2 34175.448} C_VEL
LIN {X 0,Y 712.28,Z 643.947,A -85,B 0,C 180,E1 34172.345,E2 34172.345} C_VEL
LIN {X 0,Y 712.279,Z 643.939,A -85,B 0,C 180,E1 34169.271,E2 34169.271} C_VEL
LIN {X 0,Y 712.277,Z 643.949,A -85,B 0,C 180,E1 34166.203,E2 34166.203} C_VEL
LIN {X 0,Y 712.28,Z 643.939,A -85,B 0,C 180,E1 34163.071,E2 34163.071} C_VEL
LIN {X 0,Y 712.283,Z 643.947,A -85,B 0,C 180,E1 34159.989,E2 34159.989} C_VEL
LIN {X 0,Y 712.276,Z 643.941,A -85,B 0,C 180,E1 34156.87,E2 34156.87} C_VEL
LIN {X 0,Y 712.281,Z 643.947,A -85,B 0,C 180,E1 34153.791,E2 34153.791} C_VEL
LIN {X 0,Y 712.293,Z 644.159,A -85,B 0,C 180,E1 34153.416,E2 34153.416} C_VEL
LIN {X 0,Y 713.695,Z 647.617,A -85,B 0,C 180,E1 34153.12,E2 34153.12} C_VEL
LIN {X 0,Y 718.133,Z 658.629,A -85,B 0,C 180,E1 34152.206,E2 34152.206} C_VEL
LIN {X 0,Y 716.685,Z 709.473,A -85,B 0,C 180,E1 34149.558,E2 34149.558} C_VEL
LIN {X 0,Y 716.292,Z 758.275,A -85,B 0,C 180,E1 34147.115,E2 34147.115} C_VEL
LIN {X 0,Y 718.178,Z 776.529,A -85,B 0,C 180,E1 34146.146,E2 34146.146} C_VEL
LIN {X 0,Y 721.198,Z 788.435,A -85,B 0,C 180,E1 34145.459,E2 34145.459} C_VEL
LIN {X 0,Y 725.537,Z 797.964,A -85,B 0,C 180,E1 34144.847,E2 34144.847} C_VEL
LIN {X 0,Y 731.083,Z 805.388,A -85,B 0,C 180,E1 34144.301,E2 34144.301} C_VEL
LIN {X 0,Y 736.8,Z 810.329,A -85,B 0,C 180,E1 34143.847,E2 34143.847} C_VEL
LIN {X 0,Y 740.71,Z 812.396,A -85,B 0,C 180,E1 34143.462,E2 34143.462} C_VEL
LIN {X 0,Y 744.073,Z 813.075,A -85,B 0,C 180,E1 34143.014,E2 34143.014} C_VEL
LIN {X 0,Y 746.264,Z 812.404,A -85,B 0,C 180,E1 34142.565,E2 34142.565} C_VEL
LIN {X 0,Y 747.335,Z 810.349,A -85,B 0,C 180,E1 34142.082,E2 34142.082} C_VEL
LIN {X 0,Y 746.925,Z 807.107,A -85,B 0,C 180,E1 34141.63,E2 34141.63} C_VEL
LIN {X 0,Y 745.049,Z 802.854,A -85,B 0,C 180,E1 34141.243,E2 34141.243} C_VEL
LIN {X 0,Y 741.383,Z 795.028,A -85,B 0,C 180,E1 34140.772,E2 34140.772} C_VEL
LIN {X 0,Y 738.521,Z 785.985,A -85,B 0,C 180,E1 34140.398,E2 34140.398} C_VEL
LIN {X 0,Y 736.459,Z 775.605,A -85,B 0,C 180,E1 34140.123,E2 34140.123} C_VEL
LIN {X 0,Y 735.215,Z 763.743,A -85,B 0,C 180,E1 34139.955,E2 34139.955} C_VEL
LIN {X 0,Y 734.846,Z 751.939,A -85,B 0,C 180,E1 34139.906,E2 34139.906} C_VEL
LIN {X 0,Y 734.817,Z 715.234,A -85,B 0,C 180,E1 34139.902,E2 34139.902} C_VEL
LIN {X 0,Y 730.801,Z 725.685,A -85,B 0,C 180,E1 34139.349,E2 34139.349} C_VEL
LIN {X 0,Y 727.759,Z 731.28,A -85,B 0,C 180,E1 34138.921,E2 34138.921} C_VEL
LIN {X 0,Y 725.593,Z 733.829,A -85,B 0,C 180,E1 34138.61,E2 34138.61} C_VEL
LIN {X 0,Y 721.621,Z 746.117,A -85,B 0,C 180,E1 34138.026,E2 34138.026} C_VEL
LIN {X 0,Y 718.416,Z 753.47,A -85,B 0,C 180,E1 34137.542,E2 34137.542} C_VEL
LIN {X 0,Y 716.69,Z 755.784,A -85,B 0,C 180,E1 34137.276,E2 34137.276} C_VEL
LIN {X 0,Y 715.718,Z 755.984,A -85,B 0,C 180,E1 34137.114,E2 34137.114} C_VEL
LIN {X 0,Y 715.841,Z 758.36,A -85,B 0,C 180,E1 34137.03,E2 34137.03} C_VEL
LIN {X 0,Y 716.709,Z 766.021,A -85,B 0,C 180,E1 34136.911,E2 34136.911} C_VEL
LIN {X 0,Y 715.769,Z 1033.251,A -85,B 0,C 180,E1 34134.039,E2 34134.039} C_VEL
LIN {X 0,Y 715.58,Z 1066.787,A -85,B 0,C 180,E1 34133.646,E2 34133.646} C_VEL
LIN {X 0,Y 715.372,Z 1089.049,A -85,B 0,C 180,E1 34133.231,E2 34133.231} C_VEL
LIN {X 0,Y 715.049,Z 1110.553,A -85,B 0,C 180,E1 34132.679,E2 34132.679} C_VEL
LIN {X 0,Y 714.713,Z 1131.864,A -85,B 0,C 180,E1 34131.975,E2 34131.975} C_VEL
LIN {X 0,Y 714.363,Z 1151.741,A -85,B 0,C 180,E1 34131.168,E2 34131.168} C_VEL
LIN {X 0,Y 713.944,Z 1171.595,A -85,B 0,C 180,E1 34130.194,E2 34130.194} C_VEL
LIN {X 0,Y 713.553,Z 1191.162,A -85,B 0,C 180,E1 34129.055,E2 34129.055} C_VEL
LIN {X 0,Y 713.191,Z 1209.009,A -85,B 0,C 180,E1 34127.832,E2 34127.832} C_VEL
LIN {X 0,Y 712.859,Z 1226.169,A -85,B 0,C 180,E1 34126.458,E2 34126.458} C_VEL
LIN {X 0,Y 712.577,Z 1241.242,A -85,B 0,C 180,E1 34125.044,E2 34125.044} C_VEL
LIN {X 0,Y 712.351,Z 1254.894,A -85,B 0,C 180,E1 34123.555,E2 34123.555} C_VEL
LIN {X 0,Y 712.178,Z 1267.652,A -85,B 0,C 180,E1 34121.909,E2 34121.909} C_VEL
LIN {X 0,Y 712.063,Z 1277.878,A -85,B 0,C 180,E1 34120.353,E2 34120.353} C_VEL
LIN {X 0,Y 711.981,Z 1287.536,A -85,B 0,C 180,E1 34118.56,E2 34118.56} C_VEL
LIN {X 0,Y 711.929,Z 1294.774,A -85,B 0,C 180,E1 34116.855,E2 34116.855} C_VEL
LIN {X 0,Y 711.925,Z 1300.387,A -85,B 0,C 180,E1 34115.156,E2 34115.156} C_VEL
LIN {X 0,Y 711.917,Z 1304.432,A -85,B 0,C 180,E1 34113.381,E2 34113.381} C_VEL
LIN {X 0,Y 711.909,Z 1306.765,A -85,B 0,C 180,E1 34111.609,E2 34111.609} C_VEL
LIN {X 0,Y 711.902,Z 1307.44,A -85,B 0,C 180,E1 34109.757,E2 34109.757} C_VEL
LIN {X 0,Y 711.913,Z 1306.472,A -85,B 0,C 180,E1 34108.067,E2 34108.067} C_VEL
LIN {X 0,Y 711.911,Z 1303.797,A -85,B 0,C 180,E1 34106.295,E2 34106.295} C_VEL
LIN {X 0,Y 711.922,Z 1299.396,A -85,B 0,C 180,E1 34104.519,E2 34104.519} C_VEL
LIN {X 0,Y 711.947,Z 1293.847,A -85,B 0,C 180,E1 34102.9,E2 34102.9} C_VEL
LIN {X 0,Y 711.99,Z 1286.306,A -85,B 0,C 180,E1 34101.194,E2 34101.194} C_VEL
LIN {X 0,Y 712.07,Z 1277.36,A -85,B 0,C 180,E1 34099.563,E2 34099.563} C_VEL
LIN {X 0,Y 712.178,Z 1267.633,A -85,B 0,C 180,E1 34098.088,E2 34098.088} C_VEL
LIN {X 0,Y 712.339,Z 1255.581,A -85,B 0,C 180,E1 34096.525,E2 34096.525} C_VEL
LIN {X 0,Y 712.564,Z 1242.043,A -85,B 0,C 180,E1 34095.036,E2 34095.036} C_VEL
LIN {X 0,Y 712.82,Z 1227.998,A -85,B 0,C 180,E1 34093.706,E2 34093.706} C_VEL
LIN {X 0,Y 713.161,Z 1210.599,A -85,B 0,C 180,E1 34092.286,E2 34092.286} C_VEL
LIN {X 0,Y 713.52,Z 1192.449,A -85,B 0,C 180,E1 34091.027,E2 34091.027} C_VEL
LIN {X 0,Y 713.909,Z 1173.92,A -85,B 0,C 180,E1 34089.931,E2 34089.931} C_VEL
LIN {X 0,Y 714.308,Z 1154.474,A -85,B 0,C 180,E1 34088.957,E2 34088.957} C_VEL
LIN {X 0,Y 714.659,Z 1134.043,A -85,B 0,C 180,E1 34088.107,E2 34088.107} C_VEL
LIN {X 0,Y 715.032,Z 1112.678,A -85,B 0,C 180,E1 34087.383,E2 34087.383} C_VEL
LIN {X 0,Y 715.359,Z 1090.559,A -85,B 0,C 180,E1 34086.802,E2 34086.802} C_VEL
LIN {X 0,Y 715.567,Z 1068.22,A -85,B 0,C 180,E1 34086.375,E2 34086.375} C_VEL
LIN {X 0,Y 715.757,Z 1037.178,A -85,B 0,C 180,E1 34086.003,E2 34086.003} C_VEL
LIN {X 0,Y 716.698,Z 769.108,A -85,B 0,C 180,E1 34083.123,E2 34083.123} C_VEL
LIN {X 0,Y 716.414,Z 762.161,A -85,B 0,C 180,E1 34083.035,E2 34083.035} C_VEL
LIN {X 0,Y 715.695,Z 757.296,A -85,B 0,C 180,E1 34082.95,E2 34082.95} C_VEL
LIN {X 0,Y 715.788,Z 755.823,A -85,B 0,C 180,E1 34082.864,E2 34082.864} C_VEL
LIN {X 0,Y 716.933,Z 755.587,A -85,B 0,C 180,E1 34082.686,E2 34082.686} C_VEL
LIN {X 0,Y 719.182,Z 751.983,A -85,B 0,C 180,E1 34082.341,E2 34082.341} C_VEL
LIN {X 0,Y 722.752,Z 742.95,A -85,B 0,C 180,E1 34081.806,E2 34081.806} C_VEL
LIN {X 0,Y 725.846,Z 733.364,A -85,B 0,C 180,E1 34081.354,E2 34081.354} C_VEL
LIN {X 0,Y 728.377,Z 730.344,A -85,B 0,C 180,E1 34080.991,E2 34080.991} C_VEL
LIN {X 0,Y 731.736,Z 723.527,A -85,B 0,C 180,E1 34080.521,E2 34080.521} C_VEL
LIN {X 0,Y 734.841,Z 715.164,A -85,B 0,C 180,E1 34080.095,E2 34080.095} C_VEL
LIN {X 0,Y 734.99,Z 759.338,A -85,B 0,C 180,E1 34080.075,E2 34080.075} C_VEL
LIN {X 0,Y 735.939,Z 771.752,A -85,B 0,C 180,E1 34079.947,E2 34079.947} C_VEL
LIN {X 0,Y 737.715,Z 782.538,A -85,B 0,C 180,E1 34079.71,E2 34079.71} C_VEL
LIN {X 0,Y 740.312,Z 792.077,A -85,B 0,C 180,E1 34079.367,E2 34079.367} C_VEL
LIN {X 0,Y 743.709,Z 800.329,A -85,B 0,C 180,E1 34078.928,E2 34078.928} C_VEL
LIN {X 0,Y 746.307,Z 805.413,A -85,B 0,C 180,E1 34078.543,E2 34078.543} C_VEL
LIN {X 0,Y 747.327,Z 808.922,A -85,B 0,C 180,E1 34078.141,E2 34078.141} C_VEL
LIN {X 0,Y 747.064,Z 811.365,A -85,B 0,C 180,E1 34077.721,E2 34077.721} C_VEL
LIN {X 0,Y 745.471,Z 812.844,A -85,B 0,C 180,E1 34077.245,E2 34077.245} C_VEL
LIN {X 0,Y 742.591,Z 812.933,A -85,B 0,C 180,E1 34076.768,E2 34076.768} C_VEL
LIN {X 0,Y 738.813,Z 811.541,A -85,B 0,C 180,E1 34076.339,E2 34076.339} C_VEL
LIN {X 0,Y 733.995,Z 808.204,A -85,B 0,C 180,E1 34075.92,E2 34075.92} C_VEL
LIN {X 0,Y 728.359,Z 802.117,A -85,B 0,C 180,E1 34075.365,E2 34075.365} C_VEL
LIN {X 0,Y 723.982,Z 794.467,A -85,B 0,C 180,E1 34074.778,E2 34074.778} C_VEL
LIN {X 0,Y 720.671,Z 784.678,A -85,B 0,C 180,E1 34074.122,E2 34074.122} C_VEL
LIN {X 0,Y 718.607,Z 772.674,A -85,B 0,C 180,E1 34073.404,E2 34073.404} C_VEL
LIN {X 0,Y 717.648,Z 754.314,A -85,B 0,C 180,E1 34072.391,E2 34072.391} C_VEL
LIN {X 0,Y 718.621,Z 700.981,A -85,B 0,C 180,E1 34069.561,E2 34069.561} C_VEL
LIN {X 0,Y 719.432,Z 660.65,A -85,B 0,C 180,E1 34067.346,E2 34067.346} C_VEL
LIN {X 0,Y 712.353,Z 644.441,A -85,B 0,C 180,E1 34065.945,E2 34065.945} C_VEL
LIN {X 0,Y 712.273,Z 643.947,A -85,B 0,C 180,E1 34065.87,E2 34065.87} C_VEL
LIN {X 0,Y 712.264,Z 643.947,A -85,B 0,C 180,E1 34062.911,E2 34062.911} C_VEL
LIN {X 0,Y 712.273,Z 643.946,A -85,B 0,C 180,E1 34059.907,E2 34059.907} C_VEL
LIN {X 0,Y 712.283,Z 643.948,A -85,B 0,C 180,E1 34056.929,E2 34056.929} C_VEL
LIN {X 0,Y 712.275,Z 643.948,A -85,B 0,C 180,E1 34053.937,E2 34053.937} C_VEL
LIN {X 0,Y 712.286,Z 643.993,A -85,B 0,C 180,E1 34051.622,E2 34051.622} C_VEL
LIN {X 0,Y 715.469,Z 655.125,A -85,B 0,C 180,E1 34050.578,E2 34050.578} C_VEL
LIN {X 0,Y 714.82,Z 694.027,A -85,B 0,C 180,E1 34047.491,E2 34047.491} C_VEL
LIN {X 0,Y 714.799,Z 700.565,A -85,B 0,C 180,E1 34047.004,E2 34047.004} C_VEL
LIN {X 0,Y 716.696,Z 710.01,A -85,B 0,C 180,E1 34046.822,E2 34046.822} C_VEL
LIN {X 0,Y 715.71,Z 991.672,A -85,B 0,C 180,E1 34043.798,E2 34043.798} C_VEL
LIN {X 0,Y 715.525,Z 1014.211,A -85,B 0,C 180,E1 34043.478,E2 34043.478} C_VEL
LIN {X 0,Y 715.246,Z 1036.836,A -85,B 0,C 180,E1 34043.003,E2 34043.003} C_VEL
LIN {X 0,Y 714.952,Z 1058.169,A -85,B 0,C 180,E1 34042.402,E2 34042.402} C_VEL
LIN {X 0,Y 714.588,Z 1078.429,A -85,B 0,C 180,E1 34041.679,E2 34041.679} C_VEL
LIN {X 0,Y 714.196,Z 1098.905,A -85,B 0,C 180,E1 34040.788,E2 34040.788} C_VEL
LIN {X 0,Y 713.818,Z 1118.42,A -85,B 0,C 180,E1 34039.772,E2 34039.772} C_VEL
LIN {X 0,Y 713.447,Z 1136.984,A -85,B 0,C 180,E1 34038.635,E2 34038.635} C_VEL
LIN {X 0,Y 713.071,Z 1154.392,A -85,B 0,C 180,E1 34037.378,E2 34037.378} C_VEL
LIN {X 0,Y 712.765,Z 1170.31,A -85,B 0,C 180,E1 34036.043,E2 34036.043} C_VEL
LIN {X 0,Y 712.506,Z 1185.596,A -85,B 0,C 180,E1 34034.549,E2 34034.549} C_VEL
LIN {X 0,Y 712.31,Z 1198.77,A -85,B 0,C 180,E1 34033.046,E2 34033.046} C_VEL
LIN {X 0,Y 712.148,Z 1210.434,A -85,B 0,C 180,E1 34031.47,E2 34031.47} C_VEL
LIN {X 0,Y 712.042,Z 1220.885,A -85,B 0,C 180,E1 34029.783,E2 34029.783} C_VEL
LIN {X 0,Y 711.975,Z 1229.579,A -85,B 0,C 180,E1 34028.07,E2 34028.07} C_VEL
LIN {X 0,Y 711.931,Z 1236.107,A -85,B 0,C 180,E1 34026.451,E2 34026.451} C_VEL
LIN {X 0,Y 711.915,Z 1241.283,A -85,B 0,C 180,E1 34024.753,E2 34024.753} C_VEL
LIN {X 0,Y 711.899,Z 1245.017,A -85,B 0,C 180,E1 34023,E2 34023} C_VEL
LIN {X 0,Y 711.906,Z 1246.978,A -85,B 0,C 180,E1 34021.288,E2 34021.288} C_VEL
LIN {X 0,Y 711.917,Z 1247.386,A -85,B 0,C 180,E1 34019.517,E2 34019.517} C_VEL
LIN {X 0,Y 711.903,Z 1246.182,A -85,B 0,C 180,E1 34017.746,E2 34017.746} C_VEL
LIN {X 0,Y 711.902,Z 1243.396,A -85,B 0,C 180,E1 34016.054,E2 34016.054} C_VEL
LIN {X 0,Y 711.926,Z 1238.793,A -85,B 0,C 180,E1 34014.277,E2 34014.277} C_VEL
LIN {X 0,Y 711.95,Z 1232.777,A -85,B 0,C 180,E1 34012.576,E2 34012.576} C_VEL
LIN {X 0,Y 712.002,Z 1225.296,A -85,B 0,C 180,E1 34010.951,E2 34010.951} C_VEL
LIN {X 0,Y 712.091,Z 1215.615,A -85,B 0,C 180,E1 34009.237,E2 34009.237} C_VEL
LIN {X 0,Y 712.222,Z 1205.066,A -85,B 0,C 180,E1 34007.679,E2 34007.679} C_VEL
LIN {X 0,Y 712.4,Z 1192.431,A -85,B 0,C 180,E1 34006.113,E2 34006.113} C_VEL
LIN {X 0,Y 712.629,Z 1178.33,A -85,B 0,C 180,E1 34004.622,E2 34004.622} C_VEL
LIN {X 0,Y 712.916,Z 1162.153,A -85,B 0,C 180,E1 34003.159,E2 34003.159} C_VEL
LIN {X 0,Y 713.045,Z 1156.56,A -85,B 0,C 180,E1 34002.698,E2 34002.698} C_VEL
LIN {X 0,Y 712.154,Z 1151.127,A -85,B 0,C 180,E1 34002.257,E2 34002.257} C_VEL
LIN {X 0,Y 706.434,Z 1136.858,A -85,B 0,C 180,E1 34001.074,E2 34001.074} C_VEL
LIN {X 0,Y 705.84,Z 1131.779,A -85,B 0,C 180,E1 34000.727,E2 34000.727} C_VEL
LIN {X 0,Y 706.287,Z 1113.147,A -85,B 0,C 180,E1 33999.619,E2 33999.619} C_VEL
LIN {X 0,Y 706.775,Z 1093.632,A -85,B 0,C 180,E1 33998.636,E2 33998.636} C_VEL
LIN {X 0,Y 707.182,Z 1073.345,A -85,B 0,C 180,E1 33997.792,E2 33997.792} C_VEL
LIN {X 0,Y 707.604,Z 1051.73,A -85,B 0,C 180,E1 33997.062,E2 33997.062} C_VEL
LIN {X 0,Y 707.978,Z 1029.94,A -85,B 0,C 180,E1 33996.488,E2 33996.488} C_VEL
LIN {X 0,Y 708.232,Z 1008.311,A -85,B 0,C 180,E1 33996.072,E2 33996.072} C_VEL
LIN {X 0,Y 708.434,Z 979.734,A -85,B 0,C 180,E1 33995.722,E2 33995.722} C_VEL
LIN {X 0,Y 709.539,Z 710.224,A -85,B 0,C 180,E1 33992.797,E2 33992.797} C_VEL
LIN {X 0,Y 707.24,Z 699.91,A -85,B 0,C 180,E1 33992.568,E2 33992.568} C_VEL
LIN {X 0,Y 707.96,Z 663.084,A -85,B 0,C 180,E1 33989.627,E2 33989.627} C_VEL
LIN {X 0,Y 707.843,Z 656.679,A -85,B 0,C 180,E1 33989.099,E2 33989.099} C_VEL
LIN {X 0,Y 704.334,Z 644.936,A -85,B 0,C 180,E1 33987.943,E2 33987.943} C_VEL
LIN {X 0,Y 704.333,Z 644.932,A -85,B 0,C 180,E1 33984.998,E2 33984.998} C_VEL
LIN {X 0,Y 704.341,Z 644.936,A -85,B 0,C 180,E1 33981.967,E2 33981.967} C_VEL
LIN {X 0,Y 704.343,Z 644.933,A -85,B 0,C 180,E1 33978.907,E2 33978.907} C_VEL
LIN {X 0,Y 704.341,Z 644.929,A -85,B 0,C 180,E1 33975.8,E2 33975.8} C_VEL
LIN {X 0,Y 704.336,Z 644.929,A -85,B 0,C 180,E1 33972.662,E2 33972.662} C_VEL
LIN {X 0,Y 704.345,Z 644.936,A -85,B 0,C 180,E1 33969.57,E2 33969.57} C_VEL
LIN {X 0,Y 704.334,Z 644.93,A -85,B 0,C 180,E1 33966.533,E2 33966.533} C_VEL
LIN {X 0,Y 704.329,Z 644.929,A -85,B 0,C 180,E1 33963.521,E2 33963.521} C_VEL
LIN {X 0,Y 704.326,Z 644.935,A -85,B 0,C 180,E1 33960.547,E2 33960.547} C_VEL
LIN {X 0,Y 704.32,Z 644.932,A -85,B 0,C 180,E1 33957.661,E2 33957.661} C_VEL
LIN {X 0,Y 704.329,Z 644.93,A -85,B 0,C 180,E1 33954.759,E2 33954.759} C_VEL
LIN {X 0,Y 704.338,Z 644.936,A -85,B 0,C 180,E1 33951.748,E2 33951.748} C_VEL
LIN {X 0,Y 704.343,Z 644.929,A -85,B 0,C 180,E1 33948.714,E2 33948.714} C_VEL
LIN {X 0,Y 704.339,Z 644.928,A -85,B 0,C 180,E1 33945.564,E2 33945.564} C_VEL
LIN {X 0,Y 704.341,Z 644.929,A -85,B 0,C 180,E1 33942.462,E2 33942.462} C_VEL
LIN {X 0,Y 704.339,Z 644.936,A -85,B 0,C 180,E1 33939.397,E2 33939.397} C_VEL
LIN {X 0,Y 704.336,Z 644.93,A -85,B 0,C 180,E1 33936.358,E2 33936.358} C_VEL
LIN {X 0,Y 704.334,Z 644.927,A -85,B 0,C 180,E1 33933.256,E2 33933.256} C_VEL
LIN {X 0,Y 704.346,Z 644.929,A -85,B 0,C 180,E1 33930.164,E2 33930.164} C_VEL
LIN {X 0,Y 704.328,Z 644.935,A -85,B 0,C 180,E1 33927.153,E2 33927.153} C_VEL
LIN {X 0,Y 704.319,Z 644.93,A -85,B 0,C 180,E1 33924.216,E2 33924.216} C_VEL
LIN {X 0,Y 704.323,Z 644.936,A -85,B 0,C 180,E1 33921.346,E2 33921.346} C_VEL
LIN {X 0,Y 704.332,Z 644.93,A -85,B 0,C 180,E1 33918.393,E2 33918.393} C_VEL
LIN {X 0,Y 704.34,Z 644.927,A -85,B 0,C 180,E1 33915.365,E2 33915.365} C_VEL
LIN {X 0,Y 704.338,Z 644.931,A -85,B 0,C 180,E1 33912.23,E2 33912.23} C_VEL
LIN {X 0,Y 704.341,Z 644.934,A -85,B 0,C 180,E1 33909.214,E2 33909.214} C_VEL
LIN {X 0,Y 704.338,Z 644.929,A -85,B 0,C 180,E1 33906.136,E2 33906.136} C_VEL
LIN {X 0,Y 704.342,Z 644.927,A -85,B 0,C 180,E1 33902.983,E2 33902.983} C_VEL
LIN {X 0,Y 704.34,Z 644.932,A -85,B 0,C 180,E1 33899.831,E2 33899.831} C_VEL
LIN {X 0,Y 704.332,Z 644.931,A -85,B 0,C 180,E1 33896.871,E2 33896.871} C_VEL
LIN {X 0,Y 704.324,Z 644.928,A -85,B 0,C 180,E1 33893.88,E2 33893.88} C_VEL
LIN {X 0,Y 704.331,Z 644.933,A -85,B 0,C 180,E1 33890.929,E2 33890.929} C_VEL
LIN {X 0,Y 704.338,Z 644.932,A -85,B 0,C 180,E1 33887.942,E2 33887.942} C_VEL
LIN {X 0,Y 704.326,Z 644.932,A -85,B 0,C 180,E1 33884.99,E2 33884.99} C_VEL
LIN {X 0,Y 704.332,Z 644.936,A -85,B 0,C 180,E1 33881.963,E2 33881.963} C_VEL
LIN {X 0,Y 704.361,Z 645.075,A -85,B 0,C 180,E1 33880.432,E2 33880.432} C_VEL
LIN {X 0,Y 709.051,Z 659.667,A -85,B 0,C 180,E1 33879.143,E2 33879.143} C_VEL
LIN {X 0,Y 708.309,Z 702.66,A -85,B 0,C 180,E1 33876.154,E2 33876.154} C_VEL
LIN {X 0,Y 707.344,Z 748.373,A -85,B 0,C 180,E1 33873.047,E2 33873.047} C_VEL
LIN {X 0,Y 706.457,Z 793.594,A -85,B 0,C 180,E1 33870.022,E2 33870.022} C_VEL
LIN {X 0,Y 705.707,Z 836.972,A -85,B 0,C 180,E1 33867.144,E2 33867.144} C_VEL
LIN {X 0,Y 704.994,Z 884.622,A -85,B 0,C 180,E1 33864.02,E2 33864.02} C_VEL
LIN {X 0,Y 704.954,Z 892.051,A -85,B 0,C 180,E1 33863.565,E2 33863.565} C_VEL
LIN {X 0,Y 705.356,Z 901.053,A -85,B 0,C 180,E1 33863.462,E2 33863.462} C_VEL
LIN {X 0,Y 705.03,Z 1031.942,A -85,B 0,C 180,E1 33862.098,E2 33862.098} C_VEL
LIN {X 0,Y 704.955,Z 1044.195,A -85,B 0,C 180,E1 33861.884,E2 33861.884} C_VEL
LIN {X 0,Y 704.863,Z 1056.134,A -85,B 0,C 180,E1 33861.589,E2 33861.589} C_VEL
LIN {X 0,Y 704.744,Z 1067.814,A -85,B 0,C 180,E1 33861.211,E2 33861.211} C_VEL
LIN {X 0,Y 704.618,Z 1079.458,A -85,B 0,C 180,E1 33860.736,E2 33860.736} C_VEL
LIN {X 0,Y 704.479,Z 1090.643,A -85,B 0,C 180,E1 33860.176,E2 33860.176} C_VEL
LIN {X 0,Y 704.371,Z 1101.508,A -85,B 0,C 180,E1 33859.516,E2 33859.516} C_VEL
LIN {X 0,Y 704.254,Z 1111.36,A -85,B 0,C 180,E1 33858.802,E2 33858.802} C_VEL
LIN {X 0,Y 704.162,Z 1120.284,A -85,B 0,C 180,E1 33858.032,E2 33858.032} C_VEL
LIN {X 0,Y 704.071,Z 1128.573,A -85,B 0,C 180,E1 33857.181,E2 33857.181} C_VEL
LIN {X 0,Y 704.005,Z 1136.132,A -85,B 0,C 180,E1 33856.244,E2 33856.244} C_VEL
LIN {X 0,Y 703.964,Z 1142.739,A -85,B 0,C 180,E1 33855.235,E2 33855.235} C_VEL
LIN {X 0,Y 703.935,Z 1147.974,A -85,B 0,C 180,E1 33854.225,E2 33854.225} C_VEL
LIN {X 0,Y 703.924,Z 1151.964,A -85,B 0,C 180,E1 33853.22,E2 33853.22} C_VEL
LIN {X 0,Y 703.917,Z 1155.002,A -85,B 0,C 180,E1 33852.136,E2 33852.136} C_VEL
LIN {X 0,Y 703.919,Z 1156.817,A -85,B 0,C 180,E1 33851.037,E2 33851.037} C_VEL
LIN {X 0,Y 703.917,Z 1157.406,A -85,B 0,C 180,E1 33849.98,E2 33849.98} C_VEL
LIN {X 0,Y 703.916,Z 1156.854,A -85,B 0,C 180,E1 33848.907,E2 33848.907} C_VEL
LIN {X 0,Y 703.918,Z 1155.14,A -85,B 0,C 180,E1 33847.838,E2 33847.838} C_VEL
LIN {X 0,Y 703.925,Z 1152.233,A -85,B 0,C 180,E1 33846.771,E2 33846.771} C_VEL
LIN {X 0,Y 703.935,Z 1148.072,A -85,B 0,C 180,E1 33845.706,E2 33845.706} C_VEL
LIN {X 0,Y 703.958,Z 1143.027,A -85,B 0,C 180,E1 33844.726,E2 33844.726} C_VEL
LIN {X 0,Y 703.995,Z 1137.28,A -85,B 0,C 180,E1 33843.828,E2 33843.828} C_VEL
LIN {X 0,Y 704.052,Z 1130.312,A -85,B 0,C 180,E1 33842.931,E2 33842.931} C_VEL
LIN {X 0,Y 704.126,Z 1122.745,A -85,B 0,C 180,E1 33842.116,E2 33842.116} C_VEL
LIN {X 0,Y 704.225,Z 1113.737,A -85,B 0,C 180,E1 33841.302,E2 33841.302} C_VEL
LIN {X 0,Y 704.339,Z 1104.084,A -85,B 0,C 180,E1 33840.569,E2 33840.569} C_VEL
LIN {X 0,Y 704.452,Z 1093.877,A -85,B 0,C 180,E1 33839.919,E2 33839.919} C_VEL
LIN {X 0,Y 704.561,Z 1083.197,A -85,B 0,C 180,E1 33839.349,E2 33839.349} C_VEL
LIN {X 0,Y 704.713,Z 1072.105,A -85,B 0,C 180,E1 33838.862,E2 33838.862} C_VEL
LIN {X 0,Y 704.84,Z 1059.316,A -85,B 0,C 180,E1 33838.415,E2 33838.415} C_VEL
LIN {X 0,Y 704.934,Z 1046.461,A -85,B 0,C 180,E1 33838.075,E2 33838.075} C_VEL
LIN {X 0,Y 705.014,Z 1033.471,A -85,B 0,C 180,E1 33837.833,E2 33837.833} C_VEL
LIN {X 0,Y 705.119,Z 1001.717,A -85,B 0,C 180,E1 33837.483,E2 33837.483} C_VEL
LIN {X 0,Y 705.19,Z 893.791,A -85,B 0,C 180,E1 33836.351,E2 33836.351} C_VEL
LIN {X 0,Y 705.025,Z 891.781,A -85,B 0,C 180,E1 33836.3,E2 33836.3} C_VEL
LIN {X 0,Y 705.993,Z 847.576,A -85,B 0,C 180,E1 33833.331,E2 33833.331} C_VEL
LIN {X 0,Y 707.359,Z 800.067,A -85,B 0,C 180,E1 33830.069,E2 33830.069} C_VEL
LIN {X 0,Y 708.948,Z 755.761,A -85,B 0,C 180,E1 33826.958,E2 33826.958} C_VEL
LIN {X 0,Y 710.866,Z 713.519,A -85,B 0,C 180,E1 33823.913,E2 33823.913} C_VEL
LIN {X 0,Y 711.78,Z 689.146,A -85,B 0,C 180,E1 33822.082,E2 33822.082} C_VEL
LIN {X 0,Y 712.467,Z 664.855,A -85,B 0,C 180,E1 33820.188,E2 33820.188} C_VEL
LIN {X 0,Y 707.015,Z 651.689,A -85,B 0,C 180,E1 33818.644,E2 33818.644} C_VEL
LIN {X 0,Y 705.402,Z 648.063,A -85,B 0,C 180,E1 33818.189,E2 33818.189} C_VEL
LIN {X 0,Y 704.333,Z 644.932,A -85,B 0,C 180,E1 33817.813,E2 33817.813} C_VEL
LIN {X 0,Y 704.322,Z 644.938,A -85,B 0,C 180,E1 33814.882,E2 33814.882} C_VEL
LIN {X 0,Y 704.321,Z 644.936,A -85,B 0,C 180,E1 33811.972,E2 33811.972} C_VEL
LIN {X 0,Y 704.327,Z 644.932,A -85,B 0,C 180,E1 33809.029,E2 33809.029} C_VEL
LIN {X 0,Y 704.336,Z 644.937,A -85,B 0,C 180,E1 33806.088,E2 33806.088} C_VEL
LIN {X 0,Y 704.339,Z 644.929,A -85,B 0,C 180,E1 33802.992,E2 33802.992} C_VEL
LIN {X 0,Y 704.338,Z 644.936,A -85,B 0,C 180,E1 33799.871,E2 33799.871} C_VEL
LIN {X 0,Y 704.338,Z 644.93,A -85,B 0,C 180,E1 33796.823,E2 33796.823} C_VEL
LIN {X 0,Y 704.355,Z 645.074,A -85,B 0,C 180,E1 33793.928,E2 33793.928} C_VEL
LIN {X 0,Y 705.712,Z 648.52,A -85,B 0,C 180,E1 33793.613,E2 33793.613} C_VEL
LIN {X 0,Y 711.331,Z 661.907,A -85,B 0,C 180,E1 33792.441,E2 33792.441} C_VEL
LIN {X 0,Y 709.593,Z 712.311,A -85,B 0,C 180,E1 33789.77,E2 33789.77} C_VEL
LIN {X 0,Y 709.02,Z 760.598,A -85,B 0,C 180,E1 33787.309,E2 33787.309} C_VEL
LIN {X 0,Y 710.773,Z 778.383,A -85,B 0,C 180,E1 33786.353,E2 33786.353} C_VEL
LIN {X 0,Y 713.879,Z 791.228,A -85,B 0,C 180,E1 33785.602,E2 33785.602} C_VEL
LIN {X 0,Y 718.405,Z 801.554,A -85,B 0,C 180,E1 33784.937,E2 33784.937} C_VEL
LIN {X 0,Y 723.498,Z 808.909,A -85,B 0,C 180,E1 33784.404,E2 33784.404} C_VEL
LIN {X 0,Y 730.323,Z 815.399,A -85,B 0,C 180,E1 33783.862,E2 33783.862} C_VEL
LIN {X 0,Y 735.123,Z 818.505,A -85,B 0,C 180,E1 33783.51,E2 33783.51} C_VEL
LIN {X 0,Y 739.08,Z 819.997,A -85,B 0,C 180,E1 33783.129,E2 33783.129} C_VEL
LIN {X 0,Y 742.423,Z 820.218,A -85,B 0,C 180,E1 33782.675,E2 33782.675} C_VEL
LIN {X 0,Y 744.528,Z 819.129,A -85,B 0,C 180,E1 33782.212,E2 33782.212} C_VEL
LIN {X 0,Y 745.338,Z 816.748,A -85,B 0,C 180,E1 33781.73,E2 33781.73} C_VEL
LIN {X 0,Y 744.618,Z 813.343,A -85,B 0,C 180,E1 33781.286,E2 33781.286} C_VEL
LIN {X 0,Y 742.343,Z 808.894,A -85,B 0,C 180,E1 33780.897,E2 33780.897} C_VEL
LIN {X 0,Y 738.458,Z 800.68,A -85,B 0,C 180,E1 33780.389,E2 33780.389} C_VEL
LIN {X 0,Y 735.316,Z 791.062,A -85,B 0,C 180,E1 33779.969,E2 33779.969} C_VEL
LIN {X 0,Y 732.986,Z 780.118,A -85,B 0,C 180,E1 33779.652,E2 33779.652} C_VEL
LIN {X 0,Y 731.507,Z 767.854,A -85,B 0,C 180,E1 33779.448,E2 33779.448} C_VEL
LIN {X 0,Y 730.901,Z 753.998,A -85,B 0,C 180,E1 33779.363,E2 33779.363} C_VEL
LIN {X 0,Y 730.801,Z 736.614,A -85,B 0,C 180,E1 33779.349,E2 33779.349} C_VEL
LIN {X 0,Y 728.182,Z 740.381,A -85,B 0,C 180,E1 33778.981,E2 33778.981} C_VEL
LIN {X 0,Y 724.043,Z 752.507,A -85,B 0,C 180,E1 33778.384,E2 33778.384} C_VEL
LIN {X 0,Y 720.683,Z 759.82,A -85,B 0,C 180,E1 33777.886,E2 33777.886} C_VEL
LIN {X 0,Y 718.648,Z 762.901,A -85,B 0,C 180,E1 33777.577,E2 33777.577} C_VEL
LIN {X 0,Y 714.172,Z 825.793,A -85,B 0,C 180,E1 33776.882,E2 33776.882} C_VEL
LIN {X 0,Y 711.314,Z 857.448,A -85,B 0,C 180,E1 33776.424,E2 33776.424} C_VEL
LIN {X 0,Y 709.804,Z 868.504,A -85,B 0,C 180,E1 33776.178,E2 33776.178} C_VEL
LIN {X 0,Y 709.144,Z 870.33,A -85,B 0,C 180,E1 33776.069,E2 33776.069} C_VEL
LIN {X 0,Y 708.303,Z 1063.422,A -85,B 0,C 180,E1 33773.957,E2 33773.957} C_VEL
LIN {X 0,Y 708.025,Z 1086.056,A -85,B 0,C 180,E1 33773.552,E2 33773.552} C_VEL
LIN {X 0,Y 707.646,Z 1109.097,A -85,B 0,C 180,E1 33772.974,E2 33772.974} C_VEL
LIN {X 0,Y 707.262,Z 1130.751,A -85,B 0,C 180,E1 33772.263,E2 33772.263} C_VEL
LIN {X 0,Y 706.824,Z 1151.064,A -85,B 0,C 180,E1 33771.436,E2 33771.436} C_VEL
LIN {X 0,Y 706.328,Z 1171.575,A -85,B 0,C 180,E1 33770.423,E2 33770.423} C_VEL
LIN {X 0,Y 705.867,Z 1191.169,A -85,B 0,C 180,E1 33769.271,E2 33769.271} C_VEL
LIN {X 0,Y 705.43,Z 1208.926,A -85,B 0,C 180,E1 33768.04,E2 33768.04} C_VEL
LIN {X 0,Y 705.055,Z 1225.233,A -85,B 0,C 180,E1 33766.73,E2 33766.73} C_VEL
LIN {X 0,Y 704.72,Z 1240.412,A -85,B 0,C 180,E1 33765.301,E2 33765.301} C_VEL
LIN {X 0,Y 704.463,Z 1254.192,A -85,B 0,C 180,E1 33763.794,E2 33763.794} C_VEL
LIN {X 0,Y 704.245,Z 1267.073,A -85,B 0,C 180,E1 33762.129,E2 33762.129} C_VEL
LIN {X 0,Y 704.111,Z 1276.864,A -85,B 0,C 180,E1 33760.637,E2 33760.637} C_VEL
LIN {X 0,Y 704.012,Z 1286.322,A -85,B 0,C 180,E1 33758.905,E2 33758.905} C_VEL
LIN {X 0,Y 703.96,Z 1293.849,A -85,B 0,C 180,E1 33757.179,E2 33757.179} C_VEL
LIN {X 0,Y 703.922,Z 1299.401,A -85,B 0,C 180,E1 33755.542,E2 33755.542} C_VEL
LIN {X 0,Y 703.911,Z 1303.805,A -85,B 0,C 180,E1 33753.745,E2 33753.745} C_VEL
LIN {X 0,Y 703.912,Z 1306.469,A -85,B 0,C 180,E1 33751.953,E2 33751.953} C_VEL
LIN {X 0,Y 703.902,Z 1307.44,A -85,B 0,C 180,E1 33750.243,E2 33750.243} C_VEL
LIN {X 0,Y 703.909,Z 1306.766,A -85,B 0,C 180,E1 33748.371,E2 33748.371} C_VEL
LIN {X 0,Y 703.916,Z 1304.422,A -85,B 0,C 180,E1 33746.579,E2 33746.579} C_VEL
LIN {X 0,Y 703.931,Z 1300.153,A -85,B 0,C 180,E1 33744.701,E2 33744.701} C_VEL
LIN {X 0,Y 703.944,Z 1294.466,A -85,B 0,C 180,E1 33742.983,E2 33742.983} C_VEL
LIN {X 0,Y 704.004,Z 1286.717,A -85,B 0,C 180,E1 33741.176,E2 33741.176} C_VEL
LIN {X 0,Y 704.105,Z 1277.355,A -85,B 0,C 180,E1 33739.443,E2 33739.443} C_VEL
LIN {X 0,Y 704.234,Z 1267.631,A -85,B 0,C 180,E1 33737.952,E2 33737.952} C_VEL
LIN {X 0,Y 704.43,Z 1255.585,A -85,B 0,C 180,E1 33736.371,E2 33736.371} C_VEL
LIN {X 0,Y 704.689,Z 1242.036,A -85,B 0,C 180,E1 33734.865,E2 33734.865} C_VEL
LIN {X 0,Y 705.001,Z 1227.648,A -85,B 0,C 180,E1 33733.489,E2 33733.489} C_VEL
LIN {X 0,Y 705.397,Z 1210.604,A -85,B 0,C 180,E1 33732.085,E2 33732.085} C_VEL
LIN {X 0,Y 705.829,Z 1192.455,A -85,B 0,C 180,E1 33730.812,E2 33730.812} C_VEL
LIN {X 0,Y 706.275,Z 1173.917,A -85,B 0,C 180,E1 33729.704,E2 33729.704} C_VEL
LIN {X 0,Y 706.747,Z 1154.508,A -85,B 0,C 180,E1 33728.723,E2 33728.723} C_VEL
LIN {X 0,Y 707.172,Z 1133.938,A -85,B 0,C 180,E1 33727.859,E2 33727.859} C_VEL
LIN {X 0,Y 707.6,Z 1112.322,A -85,B 0,C 180,E1 33727.121,E2 33727.121} C_VEL
LIN {X 0,Y 707.983,Z 1090.178,A -85,B 0,C 180,E1 33726.537,E2 33726.537} C_VEL
LIN {X 0,Y 708.229,Z 1068.029,A -85,B 0,C 180,E1 33726.113,E2 33726.113} C_VEL
LIN {X 0,Y 708.448,Z 1036.666,A -85,B 0,C 180,E1 33725.734,E2 33725.734} C_VEL
LIN {X 0,Y 709.183,Z 870.313,A -85,B 0,C 180,E1 33723.925,E2 33723.925} C_VEL
LIN {X 0,Y 709.899,Z 868.02,A -85,B 0,C 180,E1 33723.807,E2 33723.807} C_VEL
LIN {X 0,Y 711.549,Z 855.255,A -85,B 0,C 180,E1 33723.538,E2 33723.538} C_VEL
LIN {X 0,Y 714.553,Z 820.935,A -85,B 0,C 180,E1 33723.058,E2 33723.058} C_VEL
LIN {X 0,Y 718.718,Z 762.603,A -85,B 0,C 180,E1 33722.412,E2 33722.412} C_VEL
LIN {X 0,Y 721.399,Z 758.496,A -85,B 0,C 180,E1 33722.007,E2 33722.007} C_VEL
LIN {X 0,Y 725.009,Z 749.955,A -85,B 0,C 180,E1 33721.475,E2 33721.475} C_VEL
LIN {X 0,Y 728.498,Z 739.674,A -85,B 0,C 180,E1 33720.974,E2 33720.974} C_VEL
LIN {X 0,Y 730.886,Z 736.476,A -85,B 0,C 180,E1 33720.639,E2 33720.639} C_VEL
LIN {X 0,Y 731.067,Z 760.544,A -85,B 0,C 180,E1 33720.614,E2 33720.614} C_VEL
LIN {X 0,Y 732.059,Z 773.483,A -85,B 0,C 180,E1 33720.476,E2 33720.476} C_VEL
LIN {X 0,Y 733.867,Z 784.909,A -85,B 0,C 180,E1 33720.228,E2 33720.228} C_VEL
LIN {X 0,Y 736.519,Z 795.215,A -85,B 0,C 180,E1 33719.869,E2 33719.869} C_VEL
LIN {X 0,Y 740.057,Z 804.424,A -85,B 0,C 180,E1 33719.4,E2 33719.4} C_VEL
LIN {X 0,Y 743.882,Z 811.655,A -85,B 0,C 180,E1 33718.88,E2 33718.88} C_VEL
LIN {X 0,Y 745.211,Z 815.39,A -85,B 0,C 180,E1 33718.469,E2 33718.469} C_VEL
LIN {X 0,Y 745.081,Z 818.201,A -85,B 0,C 180,E1 33718.01,E2 33718.01} C_VEL
LIN {X 0,Y 743.62,Z 819.828,A -85,B 0,C 180,E1 33717.553,E2 33717.553} C_VEL
LIN {X 0,Y 740.84,Z 820.277,A -85,B 0,C 180,E1 33717.087,E2 33717.087} C_VEL
LIN {X 0,Y 737.169,Z 819.404,A -85,B 0,C 180,E1 33716.672,E2 33716.672} C_VEL
LIN {X 0,Y 732.963,Z 817.258,A -85,B 0,C 180,E1 33716.32,E2 33716.32} C_VEL
LIN {X 0,Y 726.627,Z 812.29,A -85,B 0,C 180,E1 33715.794,E2 33715.794} C_VEL
LIN {X 0,Y 720.953,Z 805.415,A -85,B 0,C 180,E1 33715.19,E2 33715.19} C_VEL
LIN {X 0,Y 716.392,Z 796.525,A -85,B 0,C 180,E1 33714.523,E2 33714.523} C_VEL
LIN {X 0,Y 713.119,Z 785.485,A -85,B 0,C 180,E1 33713.798,E2 33713.798} C_VEL
LIN {X 0,Y 711.19,Z 771.286,A -85,B 0,C 180,E1 33712.954,E2 33712.954} C_VEL
LIN {X 0,Y 710.684,Z 751.224,A -85,B 0,C 180,E1 33711.855,E2 33711.855} C_VEL
LIN {X 0,Y 711.813,Z 701.999,A -85,B 0,C 180,E1 33709.213,E2 33709.213} C_VEL
LIN {X 0,Y 712.735,Z 664.285,A -85,B 0,C 180,E1 33707.124,E2 33707.124} C_VEL
LIN {X 0,Y 705.189,Z 647.669,A -85,B 0,C 180,E1 33705.65,E2 33705.65} C_VEL
LIN {X 0,Y 704.337,Z 644.929,A -85,B 0,C 180,E1 33705.418,E2 33705.418} C_VEL
LIN {X 0,Y 704.327,Z 644.937,A -85,B 0,C 180,E1 33702.402,E2 33702.402} C_VEL
LIN {X 0,Y 704.344,Z 644.935,A -85,B 0,C 180,E1 33699.442,E2 33699.442} C_VEL
LIN {X 0,Y 704.322,Z 644.938,A -85,B 0,C 180,E1 33696.501,E2 33696.501} C_VEL
LIN {X 0,Y 704.327,Z 644.936,A -85,B 0,C 180,E1 33693.557,E2 33693.557} C_VEL
LIN {X 0,Y 704.355,Z 645.09,A -85,B 0,C 180,E1 33691.876,E2 33691.876} C_VEL
LIN {X 0,Y 708.024,Z 658.1,A -85,B 0,C 180,E1 33690.678,E2 33690.678} C_VEL
LIN {X 0,Y 707.319,Z 696.323,A -85,B 0,C 180,E1 33687.624,E2 33687.624} C_VEL
LIN {X 0,Y 707.323,Z 700.563,A -85,B 0,C 180,E1 33687.313,E2 33687.313} C_VEL
LIN {X 0,Y 709.551,Z 711.29,A -85,B 0,C 180,E1 33687.101,E2 33687.101} C_VEL
LIN {X 0,Y 708.387,Z 992.353,A -85,B 0,C 180,E1 33684.052,E2 33684.052} C_VEL
LIN {X 0,Y 708.17,Z 1014.686,A -85,B 0,C 180,E1 33683.729,E2 33683.729} C_VEL
LIN {X 0,Y 707.844,Z 1037.289,A -85,B 0,C 180,E1 33683.246,E2 33683.246} C_VEL
LIN {X 0,Y 707.491,Z 1058.805,A -85,B 0,C 180,E1 33682.63,E2 33682.63} C_VEL
LIN {X 0,Y 707.075,Z 1078.439,A -85,B 0,C 180,E1 33681.921,E2 33681.921} C_VEL
LIN {X 0,Y 706.636,Z 1098.501,A -85,B 0,C 180,E1 33681.041,E2 33681.041} C_VEL
LIN {X 0,Y 706.194,Z 1117.703,A -85,B 0,C 180,E1 33680.038,E2 33680.038} C_VEL
LIN {X 0,Y 705.747,Z 1135.677,A -85,B 0,C 180,E1 33678.932,E2 33678.932} C_VEL
LIN {X 0,Y 705.34,Z 1152.709,A -85,B 0,C 180,E1 33677.706,E2 33677.706} C_VEL
LIN {X 0,Y 704.959,Z 1169.391,A -85,B 0,C 180,E1 33676.31,E2 33676.31} C_VEL
LIN {X 0,Y 704.652,Z 1184.054,A -85,B 0,C 180,E1 33674.882,E2 33674.882} C_VEL
LIN {X 0,Y 704.402,Z 1197.281,A -85,B 0,C 180,E1 33673.378,E2 33673.378} C_VEL
LIN {X 0,Y 704.203,Z 1209.088,A -85,B 0,C 180,E1 33671.798,E2 33671.798} C_VEL
LIN {X 0,Y 704.08,Z 1219.968,A -85,B 0,C 180,E1 33670.06,E2 33670.06} C_VEL
LIN {X 0,Y 703.986,Z 1228.488,A -85,B 0,C 180,E1 33668.412,E2 33668.412} C_VEL
LIN {X 0,Y 703.941,Z 1235.506,A -85,B 0,C 180,E1 33666.689,E2 33666.689} C_VEL
LIN {X 0,Y 703.912,Z 1241.08,A -85,B 0,C 180,E1 33664.889,E2 33664.889} C_VEL
LIN {X 0,Y 703.901,Z 1244.797,A -85,B 0,C 180,E1 33663.176,E2 33663.176} C_VEL
LIN {X 0,Y 703.908,Z 1246.912,A -85,B 0,C 180,E1 33661.384,E2 33661.384} C_VEL
LIN {X 0,Y 703.917,Z 1247.386,A -85,B 0,C 180,E1 33659.512,E2 33659.512} C_VEL
LIN {X 0,Y 703.903,Z 1246.182,A -85,B 0,C 180,E1 33657.721,E2 33657.721} C_VEL
LIN {X 0,Y 703.902,Z 1243.394,A -85,B 0,C 180,E1 33656.009,E2 33656.009} C_VEL
LIN {X 0,Y 703.926,Z 1238.791,A -85,B 0,C 180,E1 33654.212,E2 33654.212} C_VEL
LIN {X 0,Y 703.956,Z 1232.774,A -85,B 0,C 180,E1 33652.491,E2 33652.491} C_VEL
LIN {X 0,Y 704.017,Z 1224.974,A -85,B 0,C 180,E1 33650.782,E2 33650.782} C_VEL
LIN {X 0,Y 704.126,Z 1215.612,A -85,B 0,C 180,E1 33649.113,E2 33649.113} C_VEL
LIN {X 0,Y 704.279,Z 1205.06,A -85,B 0,C 180,E1 33647.537,E2 33647.537} C_VEL
LIN {X 0,Y 704.491,Z 1192.428,A -85,B 0,C 180,E1 33645.954,E2 33645.954} C_VEL
LIN {X 0,Y 704.774,Z 1178.212,A -85,B 0,C 180,E1 33644.435,E2 33644.435} C_VEL
LIN {X 0,Y 705.114,Z 1162.216,A -85,B 0,C 180,E1 33642.973,E2 33642.973} C_VEL
LIN {X 0,Y 705.506,Z 1145.508,A -85,B 0,C 180,E1 33641.661,E2 33641.661} C_VEL
LIN {X 0,Y 705.84,Z 1131.779,A -85,B 0,C 180,E1 33640.727,E2 33640.727} C_VEL
LIN {X 0,Y 705.068,Z 1125.854,A -85,B 0,C 180,E1 33640.324,E2 33640.324} C_VEL
LIN {X 0,Y 699.722,Z 1111.073,A -85,B 0,C 180,E1 33639.298,E2 33639.298} C_VEL
LIN {X 0,Y 698.925,Z 1104.748,A -85,B 0,C 180,E1 33638.937,E2 33638.937} C_VEL
LIN {X 0,Y 699.438,Z 1084.77,A -85,B 0,C 180,E1 33638.004,E2 33638.004} C_VEL
LIN {X 0,Y 699.911,Z 1064.564,A -85,B 0,C 180,E1 33637.223,E2 33637.223} C_VEL
LIN {X 0,Y 700.379,Z 1043.345,A -85,B 0,C 180,E1 33636.562,E2 33636.562} C_VEL
LIN {X 0,Y 700.727,Z 1021.58,A -85,B 0,C 180,E1 33636.046,E2 33636.046} C_VEL
LIN {X 0,Y 701.019,Z 999.253,A -85,B 0,C 180,E1 33635.678,E2 33635.678} C_VEL
LIN {X 0,Y 702.433,Z 712.891,A -85,B 0,C 180,E1 33632.529,E2 33632.529} C_VEL
LIN {X 0,Y 700.093,Z 701.656,A -85,B 0,C 180,E1 33632.303,E2 33632.303} C_VEL
LIN {X 0,Y 699.792,Z 699.733,A -85,B 0,C 180,E1 33632.238,E2 33632.238} C_VEL
LIN {X 0,Y 700.612,Z 661.8,A -85,B 0,C 180,E1 33629.179,E2 33629.179} C_VEL
LIN {X 0,Y 700.332,Z 659.094,A -85,B 0,C 180,E1 33628.942,E2 33628.942} C_VEL
LIN {X 0,Y 696.401,Z 645.925,A -85,B 0,C 180,E1 33627.618,E2 33627.618} C_VEL
LIN {X 0,Y 696.381,Z 645.923,A -85,B 0,C 180,E1 33624.643,E2 33624.643} C_VEL
LIN {X 0,Y 696.387,Z 645.924,A -85,B 0,C 180,E1 33621.758,E2 33621.758} C_VEL
LIN {X 0,Y 696.401,Z 645.924,A -85,B 0,C 180,E1 33618.796,E2 33618.796} C_VEL
LIN {X 0,Y 696.402,Z 645.919,A -85,B 0,C 180,E1 33615.646,E2 33615.646} C_VEL
LIN {X 0,Y 696.395,Z 645.917,A -85,B 0,C 180,E1 33612.553,E2 33612.553} C_VEL
LIN {X 0,Y 696.405,Z 645.924,A -85,B 0,C 180,E1 33609.499,E2 33609.499} C_VEL
LIN {X 0,Y 696.398,Z 645.919,A -85,B 0,C 180,E1 33606.472,E2 33606.472} C_VEL
LIN {X 0,Y 696.402,Z 645.916,A -85,B 0,C 180,E1 33603.318,E2 33603.318} C_VEL
LIN {X 0,Y 696.401,Z 645.917,A -85,B 0,C 180,E1 33600.168,E2 33600.168} C_VEL
LIN {X 0,Y 696.407,Z 645.923,A -85,B 0,C 180,E1 33597.075,E2 33597.075} C_VEL
LIN {X 0,Y 696.397,Z 645.92,A -85,B 0,C 180,E1 33594.052,E2 33594.052} C_VEL
LIN {X 0,Y 696.396,Z 645.917,A -85,B 0,C 180,E1 33590.949,E2 33590.949} C_VEL
LIN {X 0,Y 696.392,Z 645.921,A -85,B 0,C 180,E1 33587.895,E2 33587.895} C_VEL
LIN {X 0,Y 696.387,Z 645.925,A -85,B 0,C 180,E1 33584.894,E2 33584.894} C_VEL
LIN {X 0,Y 696.381,Z 645.918,A -85,B 0,C 180,E1 33581.934,E2 33581.934} C_VEL
LIN {X 0,Y 696.383,Z 645.919,A -85,B 0,C 180,E1 33579.005,E2 33579.005} C_VEL
LIN {X 0,Y 696.405,Z 645.922,A -85,B 0,C 180,E1 33576.017,E2 33576.017} C_VEL
LIN {X 0,Y 696.394,Z 645.917,A -85,B 0,C 180,E1 33572.964,E2 33572.964} C_VEL
LIN {X 0,Y 696.401,Z 645.916,A -85,B 0,C 180,E1 33569.919,E2 33569.919} C_VEL
LIN {X 0,Y 696.401,Z 645.924,A -85,B 0,C 180,E1 33566.874,E2 33566.874} C_VEL
LIN {X 0,Y 696.401,Z 645.919,A -85,B 0,C 180,E1 33563.819,E2 33563.819} C_VEL
LIN {X 0,Y 696.399,Z 645.917,A -85,B 0,C 180,E1 33560.664,E2 33560.664} C_VEL
LIN {X 0,Y 696.402,Z 645.919,A -85,B 0,C 180,E1 33557.48,E2 33557.48} C_VEL
LIN {X 0,Y 696.405,Z 645.926,A -85,B 0,C 180,E1 33554.427,E2 33554.427} C_VEL
LIN {X 0,Y 696.398,Z 645.919,A -85,B 0,C 180,E1 33551.376,E2 33551.376} C_VEL
LIN {X 0,Y 696.399,Z 645.917,A -85,B 0,C 180,E1 33548.259,E2 33548.259} C_VEL
LIN {X 0,Y 696.406,Z 645.919,A -85,B 0,C 180,E1 33545.124,E2 33545.124} C_VEL
LIN {X 0,Y 696.397,Z 645.924,A -85,B 0,C 180,E1 33542.093,E2 33542.093} C_VEL
LIN {X 0,Y 696.387,Z 645.92,A -85,B 0,C 180,E1 33539.07,E2 33539.07} C_VEL
LIN {X 0,Y 696.381,Z 645.923,A -85,B 0,C 180,E1 33536.09,E2 33536.09} C_VEL
LIN {X 0,Y 696.39,Z 645.923,A -85,B 0,C 180,E1 33533.223,E2 33533.223} C_VEL
LIN {X 0,Y 696.394,Z 645.918,A -85,B 0,C 180,E1 33530.29,E2 33530.29} C_VEL
LIN {X 0,Y 696.394,Z 645.922,A -85,B 0,C 180,E1 33527.226,E2 33527.226} C_VEL
LIN {X 0,Y 696.401,Z 645.925,A -85,B 0,C 180,E1 33524.136,E2 33524.136} C_VEL
LIN {X 0,Y 696.407,Z 645.923,A -85,B 0,C 180,E1 33521.083,E2 33521.083} C_VEL
LIN {X 0,Y 696.406,Z 646.041,A -85,B 0,C 180,E1 33520.79,E2 33520.79} C_VEL
LIN {X 0,Y 701.811,Z 662.718,A -85,B 0,C 180,E1 33519.299,E2 33519.299} C_VEL
LIN {X 0,Y 700.965,Z 705.498,A -85,B 0,C 180,E1 33516.302,E2 33516.302} C_VEL
LIN {X 0,Y 699.881,Z 751.853,A -85,B 0,C 180,E1 33513.125,E2 33513.125} C_VEL
LIN {X 0,Y 698.884,Z 798.155,A -85,B 0,C 180,E1 33510.002,E2 33510.002} C_VEL
LIN {X 0,Y 698.044,Z 841.62,A -85,B 0,C 180,E1 33507.098,E2 33507.098} C_VEL
LIN {X 0,Y 697.299,Z 888.148,A -85,B 0,C 180,E1 33504.032,E2 33504.032} C_VEL
LIN {X 0,Y 697.299,Z 892.718,A -85,B 0,C 180,E1 33503.756,E2 33503.756} C_VEL
LIN {X 0,Y 697.687,Z 901.117,A -85,B 0,C 180,E1 33503.649,E2 33503.649} C_VEL
LIN {X 0,Y 697.282,Z 1029.742,A -85,B 0,C 180,E1 33502.287,E2 33502.287} C_VEL
LIN {X 0,Y 697.187,Z 1043.505,A -85,B 0,C 180,E1 33502.057,E2 33502.057} C_VEL
LIN {X 0,Y 697.074,Z 1056.004,A -85,B 0,C 180,E1 33501.748,E2 33501.748} C_VEL
LIN {X 0,Y 696.938,Z 1067.576,A -85,B 0,C 180,E1 33501.372,E2 33501.372} C_VEL
LIN {X 0,Y 696.767,Z 1080.134,A -85,B 0,C 180,E1 33500.848,E2 33500.848} C_VEL
LIN {X 0,Y 696.597,Z 1091.129,A -85,B 0,C 180,E1 33500.283,E2 33500.283} C_VEL
LIN {X 0,Y 696.461,Z 1101.613,A -85,B 0,C 180,E1 33499.63,E2 33499.63} C_VEL
LIN {X 0,Y 696.32,Z 1110.979,A -85,B 0,C 180,E1 33498.937,E2 33498.937} C_VEL
LIN {X 0,Y 696.209,Z 1119.928,A -85,B 0,C 180,E1 33498.159,E2 33498.159} C_VEL
LIN {X 0,Y 696.101,Z 1128.275,A -85,B 0,C 180,E1 33497.298,E2 33497.298} C_VEL
LIN {X 0,Y 696.025,Z 1135.931,A -85,B 0,C 180,E1 33496.343,E2 33496.343} C_VEL
LIN {X 0,Y 695.973,Z 1142.053,A -85,B 0,C 180,E1 33495.414,E2 33495.414} C_VEL
LIN {X 0,Y 695.94,Z 1147.438,A -85,B 0,C 180,E1 33494.392,E2 33494.392} C_VEL
LIN {X 0,Y 695.926,Z 1151.568,A -85,B 0,C 180,E1 33493.375,E2 33493.375} C_VEL
LIN {X 0,Y 695.917,Z 1154.738,A -85,B 0,C 180,E1 33492.278,E2 33492.278} C_VEL
LIN {X 0,Y 695.917,Z 1156.66,A -85,B 0,C 180,E1 33491.184,E2 33491.184} C_VEL
LIN {X 0,Y 695.916,Z 1157.393,A -85,B 0,C 180,E1 33490.096,E2 33490.096} C_VEL
LIN {X 0,Y 695.916,Z 1156.964,A -85,B 0,C 180,E1 33489.01,E2 33489.01} C_VEL
LIN {X 0,Y 695.918,Z 1155.375,A -85,B 0,C 180,E1 33487.928,E2 33487.928} C_VEL
LIN {X 0,Y 695.924,Z 1152.595,A -85,B 0,C 180,E1 33486.849,E2 33486.849} C_VEL
LIN {X 0,Y 695.933,Z 1148.936,A -85,B 0,C 180,E1 33485.855,E2 33485.855} C_VEL
LIN {X 0,Y 695.959,Z 1144.135,A -85,B 0,C 180,E1 33484.863,E2 33484.863} C_VEL
LIN {X 0,Y 696.003,Z 1138.073,A -85,B 0,C 180,E1 33483.872,E2 33483.872} C_VEL
LIN {X 0,Y 696.065,Z 1131.275,A -85,B 0,C 180,E1 33482.964,E2 33482.964} C_VEL
LIN {X 0,Y 696.159,Z 1123.059,A -85,B 0,C 180,E1 33482.058,E2 33482.058} C_VEL
LIN {X 0,Y 696.274,Z 1114.144,A -85,B 0,C 180,E1 33481.234,E2 33481.234} C_VEL
LIN {X 0,Y 696.421,Z 1104.75,A -85,B 0,C 180,E1 33480.494,E2 33480.494} C_VEL
LIN {X 0,Y 696.57,Z 1094.828,A -85,B 0,C 180,E1 33479.836,E2 33479.836} C_VEL
LIN {X 0,Y 696.725,Z 1083.621,A -85,B 0,C 180,E1 33479.219,E2 33479.219} C_VEL
LIN {X 0,Y 696.922,Z 1071.645,A -85,B 0,C 180,E1 33478.685,E2 33478.685} C_VEL
LIN {X 0,Y 697.074,Z 1059.453,A -85,B 0,C 180,E1 33478.253,E2 33478.253} C_VEL
LIN {X 0,Y 697.189,Z 1046.622,A -85,B 0,C 180,E1 33477.909,E2 33477.909} C_VEL
LIN {X 0,Y 697.28,Z 1033.563,A -85,B 0,C 180,E1 33477.665,E2 33477.665} C_VEL
LIN {X 0,Y 697.447,Z 999.776,A -85,B 0,C 180,E1 33477.278,E2 33477.278} C_VEL
LIN {X 0,Y 697.682,Z 948.611,A -85,B 0,C 180,E1 33476.714,E2 33476.714} C_VEL
LIN {X 0,Y 697.706,Z 894.604,A -85,B 0,C 180,E1 33476.128,E2 33476.128} C_VEL
LIN {X 0,Y 697.576,Z 893.31,A -85,B 0,C 180,E1 33476.096,E2 33476.096} C_VEL
LIN {X 0,Y 698.658,Z 849.052,A -85,B 0,C 180,E1 33473.095,E2 33473.095} C_VEL
LIN {X 0,Y 700.193,Z 800.954,A -85,B 0,C 180,E1 33469.759,E2 33469.759} C_VEL
LIN {X 0,Y 701.999,Z 756.119,A -85,B 0,C 180,E1 33466.575,E2 33466.575} C_VEL
LIN {X 0,Y 704.199,Z 712.885,A -85,B 0,C 180,E1 33463.415,E2 33463.415} C_VEL
LIN {X 0,Y 705.468,Z 681.045,A -85,B 0,C 180,E1 33460.967,E2 33460.967} C_VEL
LIN {X 0,Y 705.885,Z 668.859,A -85,B 0,C 180,E1 33459.996,E2 33459.996} C_VEL
LIN {X 0,Y 699.761,Z 653.825,A -85,B 0,C 180,E1 33458.191,E2 33458.191} C_VEL
LIN {X 0,Y 696.424,Z 646.211,A -85,B 0,C 180,E1 33457.191,E2 33457.191} C_VEL
LIN {X 0,Y 696.384,Z 645.926,A -85,B 0,C 180,E1 33456.975,E2 33456.975} C_VEL
LIN {X 0,Y 696.383,Z 645.924,A -85,B 0,C 180,E1 33454.028,E2 33454.028} C_VEL
LIN {X 0,Y 696.385,Z 645.922,A -85,B 0,C 180,E1 33451.061,E2 33451.061} C_VEL
LIN {X 0,Y 696.395,Z 645.925,A -85,B 0,C 180,E1 33448.104,E2 33448.104} C_VEL
LIN {X 0,Y 696.398,Z 645.918,A -85,B 0,C 180,E1 33445.048,E2 33445.048} C_VEL
LIN {X 0,Y 696.404,Z 645.926,A -85,B 0,C 180,E1 33441.978,E2 33441.978} C_VEL
LIN {X 0,Y 696.405,Z 645.918,A -85,B 0,C 180,E1 33438.883,E2 33438.883} C_VEL
LIN {X 0,Y 696.403,Z 645.924,A -85,B 0,C 180,E1 33435.749,E2 33435.749} C_VEL
LIN {X 0,Y 696.409,Z 646.046,A -85,B 0,C 180,E1 33434.472,E2 33434.472} C_VEL
LIN {X 0,Y 697.776,Z 649.529,A -85,B 0,C 180,E1 33434.138,E2 33434.138} C_VEL
LIN {X 0,Y 704.017,Z 663.729,A -85,B 0,C 180,E1 33432.813,E2 33432.813} C_VEL
LIN {X 0,Y 704.565,Z 665.74,A -85,B 0,C 180,E1 33432.658,E2 33432.658} C_VEL
LIN {X 0,Y 702.536,Z 715.281,A -85,B 0,C 180,E1 33429.984,E2 33429.984} C_VEL
LIN {X 0,Y 701.741,Z 761.751,A -85,B 0,C 180,E1 33427.576,E2 33427.576} C_VEL
LIN {X 0,Y 703.411,Z 780.422,A -85,B 0,C 180,E1 33426.554,E2 33426.554} C_VEL
LIN {X 0,Y 706.508,Z 793.81,A -85,B 0,C 180,E1 33425.766,E2 33425.766} C_VEL
LIN {X 0,Y 710.994,Z 804.585,A -85,B 0,C 180,E1 33425.066,E2 33425.066} C_VEL
LIN {X 0,Y 716.622,Z 813.132,A -85,B 0,C 180,E1 33424.45,E2 33424.45} C_VEL
LIN {X 0,Y 723.708,Z 820.244,A -85,B 0,C 180,E1 33423.864,E2 33423.864} C_VEL
LIN {X 0,Y 731.37,Z 825.358,A -85,B 0,C 180,E1 33423.35,E2 33423.35} C_VEL
LIN {X 0,Y 735.6,Z 827.01,A -85,B 0,C 180,E1 33422.999,E2 33422.999} C_VEL
LIN {X 0,Y 739.362,Z 827.478,A -85,B 0,C 180,E1 33422.562,E2 33422.562} C_VEL
LIN {X 0,Y 741.707,Z 826.802,A -85,B 0,C 180,E1 33422.155,E2 33422.155} C_VEL
LIN {X 0,Y 743.148,Z 824.892,A -85,B 0,C 180,E1 33421.674,E2 33421.674} C_VEL
LIN {X 0,Y 743.071,Z 821.832,A -85,B 0,C 180,E1 33421.201,E2 33421.201} C_VEL
LIN {X 0,Y 741.427,Z 817.919,A -85,B 0,C 180,E1 33420.786,E2 33420.786} C_VEL
LIN {X 0,Y 737.071,Z 809.826,A -85,B 0,C 180,E1 33420.205,E2 33420.205} C_VEL
LIN {X 0,Y 733.388,Z 800.24,A -85,B 0,C 180,E1 33419.707,E2 33419.707} C_VEL
LIN {X 0,Y 730.557,Z 789.521,A -85,B 0,C 180,E1 33419.315,E2 33419.315} C_VEL
LIN {X 0,Y 728.531,Z 777.603,A -85,B 0,C 180,E1 33419.03,E2 33419.03} C_VEL
LIN {X 0,Y 727.336,Z 764.311,A -85,B 0,C 180,E1 33418.86,E2 33418.86} C_VEL
LIN {X 0,Y 727.035,Z 757.503,A -85,B 0,C 180,E1 33418.817,E2 33418.817} C_VEL
LIN {X 0,Y 723.331,Z 765.546,A -85,B 0,C 180,E1 33418.279,E2 33418.279} C_VEL
LIN {X 0,Y 722.054,Z 767.917,A -85,B 0,C 180,E1 33418.09,E2 33418.09} C_VEL
LIN {X 0,Y 717.855,Z 826.122,A -85,B 0,C 180,E1 33417.456,E2 33417.456} C_VEL
LIN {X 0,Y 714.881,Z 858.665,A -85,B 0,C 180,E1 33416.993,E2 33416.993} C_VEL
LIN {X 0,Y 713.173,Z 871.188,A -85,B 0,C 180,E1 33416.723,E2 33416.723} C_VEL
LIN {X 0,Y 712.444,Z 874.905,A -85,B 0,C 180,E1 33416.606,E2 33416.606} C_VEL
LIN {X 0,Y 708.22,Z 943.654,A -85,B 0,C 180,E1 33415.92,E2 33415.92} C_VEL
LIN {X 0,Y 705.796,Z 962.059,A -85,B 0,C 180,E1 33415.677,E2 33415.677} C_VEL
LIN {X 0,Y 703.038,Z 975.825,A -85,B 0,C 180,E1 33415.384,E2 33415.384} C_VEL
LIN {X 0,Y 701.393,Z 983.6,A -85,B 0,C 180,E1 33415.112,E2 33415.112} C_VEL
LIN {X 0,Y 700.977,Z 1063.935,A -85,B 0,C 180,E1 33414.215,E2 33414.215} C_VEL
LIN {X 0,Y 700.661,Z 1086.422,A -85,B 0,C 180,E1 33413.807,E2 33413.807} C_VEL
LIN {X 0,Y 700.242,Z 1109.108,A -85,B 0,C 180,E1 33413.231,E2 33413.231} C_VEL
LIN {X 0,Y 699.795,Z 1130.759,A -85,B 0,C 180,E1 33412.514,E2 33412.514} C_VEL
LIN {X 0,Y 699.267,Z 1151.646,A -85,B 0,C 180,E1 33411.651,E2 33411.651} C_VEL
LIN {X 0,Y 698.724,Z 1171.593,A -85,B 0,C 180,E1 33410.654,E2 33410.654} C_VEL
LIN {X 0,Y 698.189,Z 1191.176,A -85,B 0,C 180,E1 33409.491,E2 33409.491} C_VEL
LIN {X 0,Y 697.692,Z 1208.342,A -85,B 0,C 180,E1 33408.29,E2 33408.29} C_VEL
LIN {X 0,Y 697.243,Z 1225.233,A -85,B 0,C 180,E1 33406.923,E2 33406.923} C_VEL
LIN {X 0,Y 696.857,Z 1240.404,A -85,B 0,C 180,E1 33405.477,E2 33405.477} C_VEL
LIN {X 0,Y 696.559,Z 1254.197,A -85,B 0,C 180,E1 33403.954,E2 33403.954} C_VEL
LIN {X 0,Y 696.304,Z 1267.071,A -85,B 0,C 180,E1 33402.269,E2 33402.269} C_VEL
LIN {X 0,Y 696.142,Z 1276.93,A -85,B 0,C 180,E1 33400.748,E2 33400.748} C_VEL
LIN {X 0,Y 696.031,Z 1286.326,A -85,B 0,C 180,E1 33399.007,E2 33399.007} C_VEL
LIN {X 0,Y 695.969,Z 1293.845,A -85,B 0,C 180,E1 33397.262,E2 33397.262} C_VEL
LIN {X 0,Y 695.922,Z 1299.399,A -85,B 0,C 180,E1 33395.606,E2 33395.606} C_VEL
LIN {X 0,Y 695.912,Z 1303.966,A -85,B 0,C 180,E1 33393.706,E2 33393.706} C_VEL
LIN {X 0,Y 695.913,Z 1306.546,A -85,B 0,C 180,E1 33391.893,E2 33391.893} C_VEL
LIN {X 0,Y 695.913,Z 1307.484,A -85,B 0,C 180,E1 33390.081,E2 33390.081} C_VEL
LIN {X 0,Y 695.915,Z 1306.627,A -85,B 0,C 180,E1 33388.188,E2 33388.188} C_VEL
LIN {X 0,Y 695.915,Z 1304.119,A -85,B 0,C 180,E1 33386.374,E2 33386.374} C_VEL
LIN {X 0,Y 695.925,Z 1299.646,A -85,B 0,C 180,E1 33384.475,E2 33384.475} C_VEL
LIN {X 0,Y 695.963,Z 1294.15,A -85,B 0,C 180,E1 33382.819,E2 33382.819} C_VEL
LIN {X 0,Y 696.026,Z 1286.721,A -85,B 0,C 180,E1 33381.074,E2 33381.074} C_VEL
LIN {X 0,Y 696.139,Z 1277.35,A -85,B 0,C 180,E1 33379.321,E2 33379.321} C_VEL
LIN {X 0,Y 696.292,Z 1267.629,A -85,B 0,C 180,E1 33377.813,E2 33377.813} C_VEL
LIN {X 0,Y 696.526,Z 1255.589,A -85,B 0,C 180,E1 33376.213,E2 33376.213} C_VEL
LIN {X 0,Y 696.819,Z 1242.028,A -85,B 0,C 180,E1 33374.69,E2 33374.69} C_VEL
LIN {X 0,Y 697.171,Z 1227.996,A -85,B 0,C 180,E1 33373.33,E2 33373.33} C_VEL
LIN {X 0,Y 697.651,Z 1210.193,A -85,B 0,C 180,E1 33371.848,E2 33371.848} C_VEL
LIN {X 0,Y 698.15,Z 1192.462,A -85,B 0,C 180,E1 33370.593,E2 33370.593} C_VEL
LIN {X 0,Y 698.656,Z 1173.915,A -85,B 0,C 180,E1 33369.473,E2 33369.473} C_VEL
LIN {X 0,Y 699.221,Z 1153.534,A -85,B 0,C 180,E1 33368.437,E2 33368.437} C_VEL
LIN {X 0,Y 699.729,Z 1132.938,A -85,B 0,C 180,E1 33367.57,E2 33367.57} C_VEL
LIN {X 0,Y 700.191,Z 1111.619,A -85,B 0,C 180,E1 33366.843,E2 33366.843} C_VEL
LIN {X 0,Y 700.624,Z 1089.673,A -85,B 0,C 180,E1 33366.265,E2 33366.265} C_VEL
LIN {X 0,Y 700.912,Z 1067.484,A -85,B 0,C 180,E1 33365.839,E2 33365.839} C_VEL
LIN {X 0,Y 701.159,Z 1035.348,A -85,B 0,C 180,E1 33365.451,E2 33365.451} C_VEL
LIN {X 0,Y 701.477,Z 982.597,A -85,B 0,C 180,E1 33364.863,E2 33364.863} C_VEL
LIN {X 0,Y 703.328,Z 974.5,A -85,B 0,C 180,E1 33364.579,E2 33364.579} C_VEL
LIN {X 0,Y 706.158,Z 959.94,A -85,B 0,C 180,E1 33364.289,E2 33364.289} C_VEL
LIN {X 0,Y 708.389,Z 941.467,A -85,B 0,C 180,E1 33364.056,E2 33364.056} C_VEL
LIN {X 0,Y 712.624,Z 873.587,A -85,B 0,C 180,E1 33363.365,E2 33363.365} C_VEL
LIN {X 0,Y 714.002,Z 865.957,A -85,B 0,C 180,E1 33363.145,E2 33363.145} C_VEL
LIN {X 0,Y 716.375,Z 843.524,A -85,B 0,C 180,E1 33362.773,E2 33362.773} C_VEL
LIN {X 0,Y 720.171,Z 795.483,A -85,B 0,C 180,E1 33362.192,E2 33362.192} C_VEL
LIN {X 0,Y 722.163,Z 767.472,A -85,B 0,C 180,E1 33361.893,E2 33361.893} C_VEL
LIN {X 0,Y 725.547,Z 761.057,A -85,B 0,C 180,E1 33361.397,E2 33361.397} C_VEL
LIN {X 0,Y 727.074,Z 757.605,A -85,B 0,C 180,E1 33361.177,E2 33361.177} C_VEL
LIN {X 0,Y 727.877,Z 771.691,A -85,B 0,C 180,E1 33361.062,E2 33361.062} C_VEL
LIN {X 0,Y 729.501,Z 784.096,A -85,B 0,C 180,E1 33360.833,E2 33360.833} C_VEL
LIN {X 0,Y 732.013,Z 795.57,A -85,B 0,C 180,E1 33360.482,E2 33360.482} C_VEL
LIN {X 0,Y 735.268,Z 805.553,A -85,B 0,C 180,E1 33360.038,E2 33360.038} C_VEL
LIN {X 0,Y 739.358,Z 814.385,A -85,B 0,C 180,E1 33359.492,E2 33359.492} C_VEL
LIN {X 0,Y 742.282,Z 819.616,A -85,B 0,C 180,E1 33359.053,E2 33359.053} C_VEL
LIN {X 0,Y 743.292,Z 823.079,A -85,B 0,C 180,E1 33358.627,E2 33358.627} C_VEL
LIN {X 0,Y 742.783,Z 825.737,A -85,B 0,C 180,E1 33358.149,E2 33358.149} C_VEL
LIN {X 0,Y 740.803,Z 827.215,A -85,B 0,C 180,E1 33357.666,E2 33357.666} C_VEL
LIN {X 0,Y 737.506,Z 827.398,A -85,B 0,C 180,E1 33357.202,E2 33357.202} C_VEL
LIN {X 0,Y 733.552,Z 826.329,A -85,B 0,C 180,E1 33356.818,E2 33356.818} C_VEL
LIN {X 0,Y 726.914,Z 822.718,A -85,B 0,C 180,E1 33356.325,E2 33356.325} C_VEL
LIN {X 0,Y 719.962,Z 816.926,A -85,B 0,C 180,E1 33355.725,E2 33355.725} C_VEL
LIN {X 0,Y 714.344,Z 809.843,A -85,B 0,C 180,E1 33355.11,E2 33355.11} C_VEL
LIN {X 0,Y 709.628,Z 800.573,A -85,B 0,C 180,E1 33354.413,E2 33354.413} C_VEL
LIN {X 0,Y 706.277,Z 789.378,A -85,B 0,C 180,E1 33353.663,E2 33353.663} C_VEL
LIN {X 0,Y 704.318,Z 775.773,A -85,B 0,C 180,E1 33352.838,E2 33352.838} C_VEL
LIN {X 0,Y 703.644,Z 756.723,A -85,B 0,C 180,E1 33351.772,E2 33351.772} C_VEL
LIN {X 0,Y 704.974,Z 705.327,A -85,B 0,C 180,E1 33348.987,E2 33348.987} C_VEL
LIN {X 0,Y 706.021,Z 667.885,A -85,B 0,C 180,E1 33346.898,E2 33346.898} C_VEL
LIN {X 0,Y 697.483,Z 649.043,A -85,B 0,C 180,E1 33345.204,E2 33345.204} C_VEL
LIN {X 0,Y 696.403,Z 645.913,A -85,B 0,C 180,E1 33344.916,E2 33344.916} C_VEL
LIN {X 0,Y 696.393,Z 645.925,A -85,B 0,C 180,E1 33341.948,E2 33341.948} C_VEL
LIN {X 0,Y 696.398,Z 645.922,A -85,B 0,C 180,E1 33338.862,E2 33338.862} C_VEL
LIN {X 0,Y 696.399,Z 645.925,A -85,B 0,C 180,E1 33335.759,E2 33335.759} C_VEL
LIN {X 0,Y 696.403,Z 645.926,A -85,B 0,C 180,E1 33332.714,E2 33332.714} C_VEL
LIN {X 0,Y 696.406,Z 646.106,A -85,B 0,C 180,E1 33332.162,E2 33332.162} C_VEL
LIN {X 0,Y 700.602,Z 660.597,A -85,B 0,C 180,E1 33330.821,E2 33330.821} C_VEL
LIN {X 0,Y 699.99,Z 690.038,A -85,B 0,C 180,E1 33328.45,E2 33328.45} C_VEL
LIN {X 0,Y 699.868,Z 700.595,A -85,B 0,C 180,E1 33327.629,E2 33327.629} C_VEL
LIN {X 0,Y 702.422,Z 712.805,A -85,B 0,C 180,E1 33327.382,E2 33327.382} C_VEL
LIN {X 0,Y 701.074,Z 993.695,A -85,B 0,C 180,E1 33324.304,E2 33324.304} C_VEL
LIN {X 0,Y 700.821,Z 1015.778,A -85,B 0,C 180,E1 33323.973,E2 33323.973} C_VEL
LIN {X 0,Y 700.439,Z 1038.558,A -85,B 0,C 180,E1 33323.473,E2 33323.473} C_VEL
LIN {X 0,Y 700.04,Z 1059.49,A -85,B 0,C 180,E1 33322.862,E2 33322.862} C_VEL
LIN {X 0,Y 699.56,Z 1079.445,A -85,B 0,C 180,E1 33322.129,E2 33322.129} C_VEL
LIN {X 0,Y 699.063,Z 1099.066,A -85,B 0,C 180,E1 33321.252,E2 33321.252} C_VEL
LIN {X 0,Y 698.538,Z 1118.485,A -85,B 0,C 180,E1 33320.221,E2 33320.221} C_VEL
LIN {X 0,Y 698.021,Z 1137,A -85,B 0,C 180,E1 33319.063,E2 33319.063} C_VEL
LIN {X 0,Y 697.533,Z 1154.403,A -85,B 0,C 180,E1 33317.778,E2 33317.778} C_VEL
LIN {X 0,Y 697.112,Z 1170.32,A -85,B 0,C 180,E1 33316.413,E2 33316.413} C_VEL
LIN {X 0,Y 696.739,Z 1185.611,A -85,B 0,C 180,E1 33314.885,E2 33314.885} C_VEL
LIN {X 0,Y 696.466,Z 1198.658,A -85,B 0,C 180,E1 33313.364,E2 33313.364} C_VEL
LIN {X 0,Y 696.238,Z 1210.229,A -85,B 0,C 180,E1 33311.767,E2 33311.767} C_VEL
LIN {X 0,Y 696.102,Z 1220.433,A -85,B 0,C 180,E1 33310.093,E2 33310.093} C_VEL
LIN {X 0,Y 695.992,Z 1229.218,A -85,B 0,C 180,E1 33308.343,E2 33308.343} C_VEL
LIN {X 0,Y 695.944,Z 1235.809,A -85,B 0,C 180,E1 33306.683,E2 33306.683} C_VEL
LIN {X 0,Y 695.914,Z 1241.286,A -85,B 0,C 180,E1 33304.863,E2 33304.863} C_VEL
LIN {X 0,Y 695.9,Z 1244.934,A -85,B 0,C 180,E1 33303.13,E2 33303.13} C_VEL
LIN {X 0,Y 695.906,Z 1246.979,A -85,B 0,C 180,E1 33301.317,E2 33301.317} C_VEL
LIN {X 0,Y 695.917,Z 1247.386,A -85,B 0,C 180,E1 33299.506,E2 33299.506} C_VEL
LIN {X 0,Y 695.904,Z 1246.182,A -85,B 0,C 180,E1 33297.694,E2 33297.694} C_VEL
LIN {X 0,Y 695.902,Z 1243.393,A -85,B 0,C 180,E1 33295.963,E2 33295.963} C_VEL
LIN {X 0,Y 695.926,Z 1238.79,A -85,B 0,C 180,E1 33294.145,E2 33294.145} C_VEL
LIN {X 0,Y 695.963,Z 1232.772,A -85,B 0,C 180,E1 33292.405,E2 33292.405} C_VEL
LIN {X 0,Y 696.033,Z 1225.198,A -85,B 0,C 180,E1 33290.722,E2 33290.722} C_VEL
LIN {X 0,Y 696.165,Z 1215.607,A -85,B 0,C 180,E1 33288.987,E2 33288.987} C_VEL
LIN {X 0,Y 696.335,Z 1205.053,A -85,B 0,C 180,E1 33287.393,E2 33287.393} C_VEL
LIN {X 0,Y 696.59,Z 1192.426,A -85,B 0,C 180,E1 33285.791,E2 33285.791} C_VEL
LIN {X 0,Y 696.918,Z 1178.323,A -85,B 0,C 180,E1 33284.266,E2 33284.266} C_VEL
LIN {X 0,Y 697.307,Z 1162.71,A -85,B 0,C 180,E1 33282.819,E2 33282.819} C_VEL
LIN {X 0,Y 697.761,Z 1146.102,A -85,B 0,C 180,E1 33281.494,E2 33281.494} C_VEL
LIN {X 0,Y 698.258,Z 1128.465,A -85,B 0,C 180,E1 33280.292,E2 33280.292} C_VEL
LIN {X 0,Y 698.77,Z 1109.934,A -85,B 0,C 180,E1 33279.214,E2 33279.214} C_VEL
LIN {X 0,Y 698.925,Z 1104.748,A -85,B 0,C 180,E1 33278.937,E2 33278.937} C_VEL
LIN {X 0,Y 698.137,Z 1098.308,A -85,B 0,C 180,E1 33278.585,E2 33278.585} C_VEL
LIN {X 0,Y 692.95,Z 1082.296,A -85,B 0,C 180,E1 33277.676,E2 33277.676} C_VEL
LIN {X 0,Y 692.178,Z 1075.526,A -85,B 0,C 180,E1 33277.373,E2 33277.373} C_VEL
LIN {X 0,Y 692.729,Z 1054.784,A -85,B 0,C 180,E1 33276.637,E2 33276.637} C_VEL
LIN {X 0,Y 693.209,Z 1033.236,A -85,B 0,C 180,E1 33276.035,E2 33276.035} C_VEL
LIN {X 0,Y 693.553,Z 1011.281,A -85,B 0,C 180,E1 33275.587,E2 33275.587} C_VEL
LIN {X 0,Y 693.826,Z 985.83,A -85,B 0,C 180,E1 33275.246,E2 33275.246} C_VEL
LIN {X 0,Y 695.307,Z 713.179,A -85,B 0,C 180,E1 33272.227,E2 33272.227} C_VEL
LIN {X 0,Y 692.34,Z 700.022,A -85,B 0,C 180,E1 33271.936,E2 33271.936} C_VEL
LIN {X 0,Y 693.204,Z 665.258,A -85,B 0,C 180,E1 33269.102,E2 33269.102} C_VEL
LIN {X 0,Y 692.998,Z 662.019,A -85,B 0,C 180,E1 33268.828,E2 33268.828} C_VEL
LIN {X 0,Y 688.469,Z 646.914,A -85,B 0,C 180,E1 33267.298,E2 33267.298} C_VEL
LIN {X 0,Y 688.456,Z 646.914,A -85,B 0,C 180,E1 33264.278,E2 33264.278} C_VEL
LIN {X 0,Y 688.449,Z 646.909,A -85,B 0,C 180,E1 33261.246,E2 33261.246} C_VEL
LIN {X 0,Y 688.461,Z 646.912,A -85,B 0,C 180,E1 33258.29,E2 33258.29} C_VEL
LIN {X 0,Y 688.459,Z 646.914,A -85,B 0,C 180,E1 33255.219,E2 33255.219} C_VEL
LIN {X 0,Y 688.444,Z 646.907,A -85,B 0,C 180,E1 33252.258,E2 33252.258} C_VEL
LIN {X 0,Y 688.45,Z 646.912,A -85,B 0,C 180,E1 33249.274,E2 33249.274} C_VEL
LIN {X 0,Y 688.462,Z 646.911,A -85,B 0,C 180,E1 33246.287,E2 33246.287} C_VEL
LIN {X 0,Y 688.463,Z 646.906,A -85,B 0,C 180,E1 33243.199,E2 33243.199} C_VEL
LIN {X 0,Y 688.459,Z 646.906,A -85,B 0,C 180,E1 33240.047,E2 33240.047} C_VEL
LIN {X 0,Y 688.461,Z 646.911,A -85,B 0,C 180,E1 33236.946,E2 33236.946} C_VEL
LIN {X 0,Y 688.463,Z 646.911,A -85,B 0,C 180,E1 33233.905,E2 33233.905} C_VEL
LIN {X 0,Y 688.463,Z 646.906,A -85,B 0,C 180,E1 33230.72,E2 33230.72} C_VEL
LIN {X 0,Y 688.46,Z 646.906,A -85,B 0,C 180,E1 33227.584,E2 33227.584} C_VEL
LIN {X 0,Y 688.46,Z 646.909,A -85,B 0,C 180,E1 33224.467,E2 33224.467} C_VEL
LIN {X 0,Y 688.461,Z 646.909,A -85,B 0,C 180,E1 33221.478,E2 33221.478} C_VEL
LIN {X 0,Y 688.462,Z 646.902,A -85,B 0,C 180,E1 33218.352,E2 33218.352} C_VEL
LIN {X 0,Y 688.461,Z 646.905,A -85,B 0,C 180,E1 33215.167,E2 33215.167} C_VEL
LIN {X 0,Y 688.46,Z 646.911,A -85,B 0,C 180,E1 33211.999,E2 33211.999} C_VEL
LIN {X 0,Y 688.463,Z 646.907,A -85,B 0,C 180,E1 33209.003,E2 33209.003} C_VEL
LIN {X 0,Y 688.462,Z 646.904,A -85,B 0,C 180,E1 33205.837,E2 33205.837} C_VEL
LIN {X 0,Y 688.463,Z 646.904,A -85,B 0,C 180,E1 33202.658,E2 33202.658} C_VEL
LIN {X 0,Y 688.459,Z 646.909,A -85,B 0,C 180,E1 33199.5,E2 33199.5} C_VEL
LIN {X 0,Y 688.462,Z 646.911,A -85,B 0,C 180,E1 33196.479,E2 33196.479} C_VEL
LIN {X 0,Y 688.463,Z 646.906,A -85,B 0,C 180,E1 33193.376,E2 33193.376} C_VEL
LIN {X 0,Y 688.462,Z 646.905,A -85,B 0,C 180,E1 33190.222,E2 33190.222} C_VEL
LIN {X 0,Y 688.463,Z 646.911,A -85,B 0,C 180,E1 33187.043,E2 33187.043} C_VEL
LIN {X 0,Y 688.461,Z 646.911,A -85,B 0,C 180,E1 33183.986,E2 33183.986} C_VEL
LIN {X 0,Y 688.465,Z 646.906,A -85,B 0,C 180,E1 33180.889,E2 33180.889} C_VEL
LIN {X 0,Y 688.46,Z 646.902,A -85,B 0,C 180,E1 33177.702,E2 33177.702} C_VEL
LIN {X 0,Y 688.463,Z 646.907,A -85,B 0,C 180,E1 33174.565,E2 33174.565} C_VEL
LIN {X 0,Y 688.465,Z 646.913,A -85,B 0,C 180,E1 33171.519,E2 33171.519} C_VEL
LIN {X 0,Y 688.465,Z 646.906,A -85,B 0,C 180,E1 33168.414,E2 33168.414} C_VEL
LIN {X 0,Y 688.461,Z 646.909,A -85,B 0,C 180,E1 33165.222,E2 33165.222} C_VEL
LIN {X 0,Y 688.464,Z 646.914,A -85,B 0,C 180,E1 33162.088,E2 33162.088} C_VEL
LIN {X 0,Y 688.486,Z 647.078,A -85,B 0,C 180,E1 33161.15,E2 33161.15} C_VEL
LIN {X 0,Y 694.572,Z 665.589,A -85,B 0,C 180,E1 33159.468,E2 33159.468} C_VEL
LIN {X 0,Y 693.666,Z 707.164,A -85,B 0,C 180,E1 33156.536,E2 33156.536} C_VEL
LIN {X 0,Y 692.477,Z 752.834,A -85,B 0,C 180,E1 33153.377,E2 33153.377} C_VEL
LIN {X 0,Y 691.391,Z 798.582,A -85,B 0,C 180,E1 33150.265,E2 33150.265} C_VEL
LIN {X 0,Y 690.45,Z 843.635,A -85,B 0,C 180,E1 33147.234,E2 33147.234} C_VEL
LIN {X 0,Y 689.641,Z 889.63,A -85,B 0,C 180,E1 33144.179,E2 33144.179} C_VEL
LIN {X 0,Y 689.658,Z 893.445,A -85,B 0,C 180,E1 33143.955,E2 33143.955} C_VEL
LIN {X 0,Y 690.062,Z 901.409,A -85,B 0,C 180,E1 33143.847,E2 33143.847} C_VEL
LIN {X 0,Y 689.549,Z 1028.201,A -85,B 0,C 180,E1 33142.476,E2 33142.476} C_VEL
LIN {X 0,Y 689.439,Z 1043.695,A -85,B 0,C 180,E1 33142.222,E2 33142.222} C_VEL
LIN {X 0,Y 689.31,Z 1057.04,A -85,B 0,C 180,E1 33141.888,E2 33141.888} C_VEL
LIN {X 0,Y 689.137,Z 1070.074,A -85,B 0,C 180,E1 33141.447,E2 33141.447} C_VEL
LIN {X 0,Y 688.948,Z 1082.276,A -85,B 0,C 180,E1 33140.918,E2 33140.918} C_VEL
LIN {X 0,Y 688.763,Z 1093.477,A -85,B 0,C 180,E1 33140.319,E2 33140.319} C_VEL
LIN {X 0,Y 688.604,Z 1103.935,A -85,B 0,C 180,E1 33139.643,E2 33139.643} C_VEL
LIN {X 0,Y 688.439,Z 1113.571,A -85,B 0,C 180,E1 33138.898,E2 33138.898} C_VEL
LIN {X 0,Y 688.298,Z 1122.136,A -85,B 0,C 180,E1 33138.112,E2 33138.112} C_VEL
LIN {X 0,Y 688.166,Z 1130.102,A -85,B 0,C 180,E1 33137.242,E2 33137.242} C_VEL
LIN {X 0,Y 688.074,Z 1136.744,A -85,B 0,C 180,E1 33136.375,E2 33136.375} C_VEL
LIN {X 0,Y 688.002,Z 1142.753,A -85,B 0,C 180,E1 33135.424,E2 33135.424} C_VEL
LIN {X 0,Y 687.954,Z 1147.963,A -85,B 0,C 180,E1 33134.391,E2 33134.391} C_VEL
LIN {X 0,Y 687.933,Z 1151.944,A -85,B 0,C 180,E1 33133.362,E2 33133.362} C_VEL
LIN {X 0,Y 687.921,Z 1154.808,A -85,B 0,C 180,E1 33132.337,E2 33132.337} C_VEL
LIN {X 0,Y 687.917,Z 1156.722,A -85,B 0,C 180,E1 33131.231,E2 33131.231} C_VEL
LIN {X 0,Y 687.916,Z 1157.475,A -85,B 0,C 180,E1 33130.13,E2 33130.13} C_VEL
LIN {X 0,Y 687.917,Z 1157.094,A -85,B 0,C 180,E1 33129.032,E2 33129.032} C_VEL
LIN {X 0,Y 687.92,Z 1155.583,A -85,B 0,C 180,E1 33127.937,E2 33127.937} C_VEL
LIN {X 0,Y 687.93,Z 1152.916,A -85,B 0,C 180,E1 33126.845,E2 33126.845} C_VEL
LIN {X 0,Y 687.952,Z 1149.034,A -85,B 0,C 180,E1 33125.756,E2 33125.756} C_VEL
LIN {X 0,Y 687.994,Z 1144.3,A -85,B 0,C 180,E1 33124.752,E2 33124.752} C_VEL
LIN {X 0,Y 688.066,Z 1138.328,A -85,B 0,C 180,E1 33123.749,E2 33123.749} C_VEL
LIN {X 0,Y 688.165,Z 1131.628,A -85,B 0,C 180,E1 33122.832,E2 33122.832} C_VEL
LIN {X 0,Y 688.304,Z 1123.529,A -85,B 0,C 180,E1 33121.915,E2 33121.915} C_VEL
LIN {X 0,Y 688.462,Z 1114.682,A -85,B 0,C 180,E1 33121.082,E2 33121.082} C_VEL
LIN {X 0,Y 688.633,Z 1105.222,A -85,B 0,C 180,E1 33120.333,E2 33120.333} C_VEL
LIN {X 0,Y 688.811,Z 1094.522,A -85,B 0,C 180,E1 33119.626,E2 33119.626} C_VEL
LIN {X 0,Y 688.982,Z 1083.919,A -85,B 0,C 180,E1 33119.044,E2 33119.044} C_VEL
LIN {X 0,Y 689.197,Z 1071.816,A -85,B 0,C 180,E1 33118.504,E2 33118.504} C_VEL
LIN {X 0,Y 689.363,Z 1059.443,A -85,B 0,C 180,E1 33118.067,E2 33118.067} C_VEL
LIN {X 0,Y 689.491,Z 1045.972,A -85,B 0,C 180,E1 33117.712,E2 33117.712} C_VEL
LIN {X 0,Y 689.585,Z 1032.15,A -85,B 0,C 180,E1 33117.465,E2 33117.465} C_VEL
LIN {X 0,Y 689.81,Z 990.214,A -85,B 0,C 180,E1 33116.985,E2 33116.985} C_VEL
LIN {X 0,Y 690.299,Z 911.462,A -85,B 0,C 180,E1 33116.096,E2 33116.096} C_VEL
LIN {X 0,Y 690.216,Z 895.219,A -85,B 0,C 180,E1 33115.89,E2 33115.89} C_VEL
LIN {X 0,Y 691.226,Z 854.189,A -85,B 0,C 180,E1 33113.104,E2 33113.104} C_VEL
LIN {X 0,Y 692.758,Z 809.539,A -85,B 0,C 180,E1 33109.984,E2 33109.984} C_VEL
LIN {X 0,Y 694.565,Z 766.944,A -85,B 0,C 180,E1 33106.937,E2 33106.937} C_VEL
LIN {X 0,Y 696.907,Z 723.607,A -85,B 0,C 180,E1 33103.753,E2 33103.753} C_VEL
LIN {X 0,Y 698.074,Z 701.421,A -85,B 0,C 180,E1 33102.064,E2 33102.064} C_VEL
LIN {X 0,Y 699.333,Z 672.874,A -85,B 0,C 180,E1 33099.8,E2 33099.8} C_VEL
LIN {X 0,Y 693.251,Z 658.149,A -85,B 0,C 180,E1 33097.975,E2 33097.975} C_VEL
LIN {X 0,Y 689.718,Z 650.347,A -85,B 0,C 180,E1 33096.912,E2 33096.912} C_VEL
LIN {X 0,Y 688.459,Z 646.914,A -85,B 0,C 180,E1 33096.434,E2 33096.434} C_VEL
LIN {X 0,Y 688.458,Z 646.908,A -85,B 0,C 180,E1 33093.334,E2 33093.334} C_VEL
LIN {X 0,Y 688.462,Z 646.913,A -85,B 0,C 180,E1 33090.282,E2 33090.282} C_VEL
LIN {X 0,Y 688.463,Z 646.907,A -85,B 0,C 180,E1 33087.199,E2 33087.199} C_VEL
LIN {X 0,Y 688.461,Z 646.915,A -85,B 0,C 180,E1 33084.073,E2 33084.073} C_VEL
LIN {X 0,Y 688.465,Z 646.906,A -85,B 0,C 180,E1 33080.926,E2 33080.926} C_VEL
LIN {X 0,Y 688.46,Z 646.913,A -85,B 0,C 180,E1 33077.788,E2 33077.788} C_VEL
LIN {X 0,Y 688.475,Z 647.119,A -85,B 0,C 180,E1 33075.068,E2 33075.068} C_VEL
LIN {X 0,Y 689.738,Z 650.35,A -85,B 0,C 180,E1 33074.737,E2 33074.737} C_VEL
LIN {X 0,Y 693.802,Z 658.944,A -85,B 0,C 180,E1 33073.837,E2 33073.837} C_VEL
LIN {X 0,Y 697.854,Z 668.704,A -85,B 0,C 180,E1 33072.931,E2 33072.931} C_VEL
LIN {X 0,Y 695.613,Z 715.768,A -85,B 0,C 180,E1 33070.34,E2 33070.34} C_VEL
LIN {X 0,Y 694.542,Z 764.25,A -85,B 0,C 180,E1 33067.78,E2 33067.78} C_VEL
LIN {X 0,Y 696.189,Z 783.067,A -85,B 0,C 180,E1 33066.734,E2 33066.734} C_VEL
LIN {X 0,Y 699.083,Z 796.136,A -85,B 0,C 180,E1 33065.948,E2 33065.948} C_VEL
LIN {X 0,Y 703.21,Z 806.776,A -85,B 0,C 180,E1 33065.258,E2 33065.258} C_VEL
LIN {X 0,Y 708.447,Z 815.593,A -85,B 0,C 180,E1 33064.63,E2 33064.63} C_VEL
LIN {X 0,Y 714.578,Z 822.714,A -85,B 0,C 180,E1 33064.068,E2 33064.068} C_VEL
LIN {X 0,Y 722.025,Z 828.8,A -85,B 0,C 180,E1 33063.521,E2 33063.521} C_VEL
LIN {X 0,Y 729.114,Z 832.859,A -85,B 0,C 180,E1 33063.078,E2 33063.078} C_VEL
LIN {X 0,Y 733.416,Z 834.315,A -85,B 0,C 180,E1 33062.735,E2 33062.735} C_VEL
LIN {X 0,Y 737.319,Z 834.611,A -85,B 0,C 180,E1 33062.295,E2 33062.295} C_VEL
LIN {X 0,Y 740.057,Z 833.554,A -85,B 0,C 180,E1 33061.805,E2 33061.805} C_VEL
LIN {X 0,Y 741.24,Z 831.415,A -85,B 0,C 180,E1 33061.332,E2 33061.332} C_VEL
LIN {X 0,Y 740.914,Z 828.282,A -85,B 0,C 180,E1 33060.873,E2 33060.873} C_VEL
LIN {X 0,Y 739.023,Z 824.323,A -85,B 0,C 180,E1 33060.465,E2 33060.465} C_VEL
LIN {X 0,Y 734.444,Z 815.936,A -85,B 0,C 180,E1 33059.851,E2 33059.851} C_VEL
LIN {X 0,Y 730.557,Z 806.037,A -85,B 0,C 180,E1 33059.315,E2 33059.315} C_VEL
LIN {X 0,Y 727.457,Z 794.845,A -85,B 0,C 180,E1 33058.877,E2 33058.877} C_VEL
LIN {X 0,Y 725.205,Z 782.574,A -85,B 0,C 180,E1 33058.553,E2 33058.553} C_VEL
LIN {X 0,Y 724.981,Z 781.384,A -85,B 0,C 180,E1 33058.521,E2 33058.521} C_VEL
LIN {X 0,Y 720.8,Z 836.074,A -85,B 0,C 180,E1 33057.903,E2 33057.903} C_VEL
LIN {X 0,Y 718.027,Z 864.129,A -85,B 0,C 180,E1 33057.482,E2 33057.482} C_VEL
LIN {X 0,Y 716.347,Z 875.136,A -85,B 0,C 180,E1 33057.223,E2 33057.223} C_VEL
LIN {X 0,Y 715.92,Z 877.918,A -85,B 0,C 180,E1 33057.156,E2 33057.156} C_VEL
LIN {X 0,Y 712.399,Z 931.17,A -85,B 0,C 180,E1 33056.65,E2 33056.65} C_VEL
LIN {X 0,Y 709.17,Z 950.791,A -85,B 0,C 180,E1 33056.478,E2 33056.478} C_VEL
LIN {X 0,Y 704.849,Z 968.225,A -85,B 0,C 180,E1 33056.234,E2 33056.234} C_VEL
LIN {X 0,Y 701.6,Z 980.153,A -85,B 0,C 180,E1 33055.944,E2 33055.944} C_VEL
LIN {X 0,Y 700.035,Z 986.269,A -85,B 0,C 180,E1 33055.734,E2 33055.734} C_VEL
LIN {X 0,Y 696.687,Z 997.271,A -85,B 0,C 180,E1 33055.502,E2 33055.502} C_VEL
LIN {X 0,Y 694.297,Z 1006.376,A -85,B 0,C 180,E1 33055.185,E2 33055.185} C_VEL
LIN {X 0,Y 694.023,Z 1008.666,A -85,B 0,C 180,E1 33055.117,E2 33055.117} C_VEL
LIN {X 0,Y 693.667,Z 1064.272,A -85,B 0,C 180,E1 33054.481,E2 33054.481} C_VEL
LIN {X 0,Y 693.31,Z 1086.787,A -85,B 0,C 180,E1 33054.067,E2 33054.067} C_VEL
LIN {X 0,Y 692.853,Z 1109.102,A -85,B 0,C 180,E1 33053.493,E2 33053.493} C_VEL
LIN {X 0,Y 692.341,Z 1130.766,A -85,B 0,C 180,E1 33052.769,E2 33052.769} C_VEL
LIN {X 0,Y 691.737,Z 1151.722,A -85,B 0,C 180,E1 33051.895,E2 33051.895} C_VEL
LIN {X 0,Y 691.134,Z 1171.59,A -85,B 0,C 180,E1 33050.891,E2 33050.891} C_VEL
LIN {X 0,Y 690.521,Z 1191.183,A -85,B 0,C 180,E1 33049.716,E2 33049.716} C_VEL
LIN {X 0,Y 689.951,Z 1208.331,A -85,B 0,C 180,E1 33048.503,E2 33048.503} C_VEL
LIN {X 0,Y 689.446,Z 1225.233,A -85,B 0,C 180,E1 33047.12,E2 33047.12} C_VEL
LIN {X 0,Y 689.002,Z 1240.396,A -85,B 0,C 180,E1 33045.658,E2 33045.658} C_VEL
LIN {X 0,Y 688.655,Z 1254.201,A -85,B 0,C 180,E1 33044.117,E2 33044.117} C_VEL
LIN {X 0,Y 688.363,Z 1267.07,A -85,B 0,C 180,E1 33042.413,E2 33042.413} C_VEL
LIN {X 0,Y 688.174,Z 1276.853,A -85,B 0,C 180,E1 33040.886,E2 33040.886} C_VEL
